LIN {X -0.027,Y -225.193,Z 1512.224,A 0.000,B 0.000,C 90.000,E1 40.334} C_DIS
LIN {X 0.094,Y -218.602,Z 1512.207,A 0.000,B 0.000,C 90.000,E1 37.237} C_DIS
LIN {X 0.128,Y -212.681,Z 1512.190,A 0.000,B 0.000,C 90.000,E1 34.119} C_DIS
LIN {X 0.027,Y -206.125,Z 1512.168,A 0.000,B 0.000,C 90.000,E1 30.207} C_DIS
LIN {X -0.041,Y -200.324,Z 1512.146,A 0.000,B 0.000,C 90.000,E1 26.232} C_DIS
LIN {X 0.082,Y -195.443,Z 1512.123,A 0.000,B 0.000,C 90.000,E1 22.153} C_DIS
LIN {X -0.062,Y -191.314,Z 1512.100,A 0.000,B 0.000,C 90.000,E1 18.109} C_DIS
LIN {X 0.065,Y -187.294,Z 1512.073,A 0.000,B 0.000,C 90.000,E1 13.119} C_DIS
LIN {X 0.047,Y -183.991,Z 1512.041,A 0.000,B 0.000,C 90.000,E1 7.296} C_DIS
LIN {X 0.026,Y -182.029,Z 1511.993,A 0.000,B 0.000,C 90.000,E1 358.682} C_DIS
LIN {X -0.047,Y -182.890,Z 1511.951,A 0.000,B 0.000,C 90.000,E1 351.141} C_DIS
LIN {X -0.073,Y -185.382,Z 1511.918,A 0.000,B 0.000,C 90.000,E1 345.283} C_DIS
LIN {X 0.069,Y -188.835,Z 1511.890,A 0.000,B 0.000,C 90.000,E1 340.242} C_DIS
LIN {X 0.097,Y -192.632,Z 1511.867,A 0.000,B 0.000,C 90.000,E1 336.102} C_DIS
LIN {X 0.032,Y -197.354,Z 1511.845,A 0.000,B 0.000,C 90.000,E1 332.025} C_DIS
LIN {X -0.004,Y -201.753,Z 1511.827,A 0.000,B 0.000,C 90.000,E1 328.791} C_DIS
LIN {X -0.067,Y -206.915,Z 1511.809,A 0.000,B 0.000,C 90.000,E1 325.595} C_DIS
LIN {X 0.012,Y -212.787,Z 1511.791,A 0.000,B 0.000,C 90.000,E1 322.396} C_DIS
LIN {X 0.031,Y -219.487,Z 1511.774,A 0.000,B 0.000,C 90.000,E1 319.256} C_DIS
LIN {X -0.081,Y -228.037,Z 1511.754,A 0.000,B 0.000,C 90.000,E1 315.810} C_DIS
LIN {X -0.043,Y -236.681,Z 1511.738,A 0.000,B 0.000,C 90.000,E1 312.771} C_DIS
LIN {X -0.083,Y -246.539,Z 1511.721,A 0.000,B 0.000,C 90.000,E1 309.806} C_DIS
LIN {X -0.058,Y -253.422,Z 1511.711,A 0.000,B 0.000,C 90.000,E1 307.971} C_DIS
LIN {X -0.074,Y -261.276,Z 1511.701,A 0.000,B 0.000,C 90.000,E1 306.171} C_DIS
LIN {X -0.032,Y -268.244,Z 1511.693,A 0.000,B 0.000,C 90.000,E1 304.739} C_DIS
LIN {X 0.169,Y -275.984,Z 1511.685,A 0.000,B 0.000,C 90.000,E1 303.293} C_DIS
LIN {X 0.012,Y -288.868,Z 1511.674,A 0.000,B 0.000,C 90.000,E1 301.258} C_DIS
LIN {X -0.059,Y -303.145,Z 1511.662,A 0.000,B 0.000,C 90.000,E1 299.255} C_DIS
LIN {X 0.162,Y -318.859,Z 1511.652,A 0.000,B 0.000,C 90.000,E1 297.257} C_DIS
LIN {X 0.039,Y -342.911,Z 1511.637,A 0.000,B 0.000,C 90.000,E1 294.591} C_DIS
LIN {X 0.109,Y -358.996,Z 1511.627,A 0.000,B 0.000,C 90.000,E1 292.898} C_DIS
LIN {X 0.010,Y -372.297,Z 1511.620,A 0.000,B 0.000,C 90.000,E1 291.535} C_DIS
LIN {X 0.017,Y -382.747,Z 1511.614,A 0.000,B 0.000,C 90.000,E1 290.429} C_DIS
LIN {X -0.118,Y -392.921,Z 1511.607,A 0.000,B 0.000,C 90.000,E1 289.322} C_DIS
LIN {X -0.060,Y -402.520,Z 1511.601,A 0.000,B 0.000,C 90.000,E1 288.181} C_DIS
LIN {X 0.022,Y -409.127,Z 1511.596,A 0.000,B 0.000,C 90.000,E1 287.330} C_DIS
LIN {X 0.049,Y -415.053,Z 1511.592,A 0.000,B 0.000,C 90.000,E1 286.496} C_DIS
LIN {X 0.127,Y -420.270,Z 1511.587,A 0.000,B 0.000,C 90.000,E1 285.662} C_DIS
LIN {X 0.000,Y -423.330,Z 1511.584,A 0.000,B 0.000,C 90.000,E1 285.134} C_DIS
LIN {X 0.162,Y -427.242,Z 1511.580,A 0.000,B 0.000,C 90.000,E1 284.300} C_DIS
LIN {X -0.166,Y -430.462,Z 1511.575,A 0.000,B 0.000,C 90.000,E1 283.536} C_DIS
LIN {X -0.227,Y -432.118,Z 1511.572,A 0.000,B 0.000,C 90.000,E1 283.008} C_DIS
LIN {X 0.234,Y -433.418,Z 1511.569,A 0.000,B 0.000,C 90.000,E1 282.411} C_DIS
LIN {X 0.098,Y -434.287,Z 1511.566,A 0.000,B 0.000,C 90.000,E1 281.895} C_DIS
LIN {X 0.060,Y -434.706,Z 1511.563,A 0.000,B 0.000,C 90.000,E1 281.366} C_DIS
LIN {X 0.027,Y -434.628,Z 1511.560,A 0.000,B 0.000,C 90.000,E1 280.838} C_DIS
LIN {X -0.006,Y -433.917,Z 1511.557,A 0.000,B 0.000,C 90.000,E1 280.310} C_DIS
LIN {X -0.116,Y -432.707,Z 1511.554,A 0.000,B 0.000,C 90.000,E1 279.792} C_DIS
LIN {X -0.155,Y -430.824,Z 1511.551,A 0.000,B 0.000,C 90.000,E1 279.265} C_DIS
LIN {X 0.154,Y -428.183,Z 1511.548,A 0.000,B 0.000,C 90.000,E1 278.690} C_DIS
LIN {X 0.083,Y -424.707,Z 1511.545,A 0.000,B 0.000,C 90.000,E1 278.163} C_DIS
LIN {X -0.065,Y -420.373,Z 1511.542,A 0.000,B 0.000,C 90.000,E1 277.644} C_DIS
LIN {X 0.182,Y -414.947,Z 1511.539,A 0.000,B 0.000,C 90.000,E1 277.068} C_DIS
LIN {X -0.099,Y -408.967,Z 1511.537,A 0.000,B 0.000,C 90.000,E1 276.606} C_DIS
LIN {X -0.009,Y -402.725,Z 1511.534,A 0.000,B 0.000,C 90.000,E1 276.144} C_DIS
LIN {X 0.054,Y -396.391,Z 1511.532,A 0.000,B 0.000,C 90.000,E1 275.739} C_DIS
LIN {X -0.021,Y -389.878,Z 1511.530,A 0.000,B 0.000,C 90.000,E1 275.391} C_DIS
LIN {X 0.072,Y -383.135,Z 1511.528,A 0.000,B 0.000,C 90.000,E1 275.049} C_DIS
LIN {X -0.084,Y -373.272,Z 1511.526,A 0.000,B 0.000,C 90.000,E1 274.645} C_DIS
LIN {X -0.080,Y -357.522,Z 1511.522,A 0.000,B 0.000,C 90.000,E1 274.012} C_DIS
LIN {X 0.125,Y -344.511,Z 1511.520,A 0.000,B 0.000,C 90.000,E1 273.498} C_DIS
LIN {X -0.002,Y -331.363,Z 1511.517,A 0.000,B 0.000,C 90.000,E1 273.094} C_DIS
LIN {X 0.011,Y -321.220,Z 1511.516,A 0.000,B 0.000,C 90.000,E1 272.808} C_DIS
LIN {X 0.022,Y -314.381,Z 1511.515,A 0.000,B 0.000,C 90.000,E1 272.636} C_DIS
LIN {X 0.092,Y -302.749,Z 1511.513,A 0.000,B 0.000,C 90.000,E1 272.407} C_DIS
LIN {X 0.053,Y -294.444,Z 1511.513,A 0.000,B 0.000,C 90.000,E1 272.293} C_DIS
LIN {X -0.020,Y -280.477,Z 1511.512,A 0.000,B 0.000,C 90.000,E1 272.178} C_DIS
LIN {X -0.124,Y -275.438,Z 1511.512,A 0.000,B 0.000,C 90.000,E1 272.178} C_DIS
LIN {X 0.066,Y -181.239,Z 1511.512,A 0.000,B 0.000,C 90.000,E1 272.121} C_DIS
LIN {X 0.075,Y -181.574,Z 1511.502,A 0.000,B 0.000,C 90.000,E1 270.401} C_DIS
LIN {X 0.051,Y -180.906,Z 1511.474,A 0.000,B 0.000,C 90.000,E1 265.355} C_DIS
LIN {X -0.055,Y -180.690,Z 1511.470,A 0.000,B 0.000,C 90.000,E1 264.546} C_DIS
LIN {X 0.024,Y -178.774,Z 1511.441,A 0.000,B 0.000,C 90.000,E1 259.454} C_DIS
LIN {X -0.074,Y -175.820,Z 1511.413,A 0.000,B 0.000,C 90.000,E1 254.393} C_DIS
LIN {X -0.073,Y -172.007,Z 1511.385,A 0.000,B 0.000,C 90.000,E1 249.263} C_DIS
LIN {X -0.096,Y -171.426,Z 1511.380,A 0.000,B 0.000,C 90.000,E1 248.411} C_DIS
LIN {X -0.041,Y -167.663,Z 1511.356,A 0.000,B 0.000,C 90.000,E1 244.076} C_DIS
LIN {X -0.100,Y -166.333,Z 1511.346,A 0.000,B 0.000,C 90.000,E1 242.359} C_DIS
LIN {X 0.032,Y -163.072,Z 1511.327,A 0.000,B 0.000,C 90.000,E1 238.820} C_DIS
LIN {X -0.056,Y -161.011,Z 1511.312,A 0.000,B 0.000,C 90.000,E1 236.215} C_DIS
LIN {X 0.054,Y -157.754,Z 1511.292,A 0.000,B 0.000,C 90.000,E1 232.637} C_DIS
LIN {X -0.007,Y -155.792,Z 1511.278,A 0.000,B 0.000,C 90.000,E1 229.989} C_DIS
LIN {X 0.047,Y -152.046,Z 1511.253,A 0.000,B 0.000,C 90.000,E1 225.486} C_DIS
LIN {X 0.064,Y -150.295,Z 1511.238,A 0.000,B 0.000,C 90.000,E1 222.771} C_DIS
LIN {X -0.010,Y -147.041,Z 1511.213,A 0.000,B 0.000,C 90.000,E1 218.257} C_DIS
LIN {X -0.018,Y -145.622,Z 1511.197,A 0.000,B 0.000,C 90.000,E1 215.518} C_DIS
LIN {X -0.018,Y -143.006,Z 1511.172,A 0.000,B 0.000,C 90.000,E1 210.924} C_DIS
LIN {X 0.039,Y -141.632,Z 1511.151,A 0.000,B 0.000,C 90.000,E1 207.206} C_DIS
LIN {X -0.036,Y -139.436,Z 1511.115,A 0.000,B 0.000,C 90.000,E1 200.737} C_DIS
LIN {X 0.018,Y -139.167,Z 1511.105,A 0.000,B 0.000,C 90.000,E1 198.852} C_DIS
LIN {X 0.051,Y -138.316,Z 1511.053,A 0.000,B 0.000,C 90.000,E1 189.500} C_DIS
LIN {X 0.063,Y -139.475,Z 1511.006,A 0.000,B 0.000,C 90.000,E1 181.088} C_DIS
LIN {X 0.004,Y -141.054,Z 1510.975,A 0.000,B 0.000,C 90.000,E1 175.527} C_DIS
LIN {X -0.042,Y -142.426,Z 1510.960,A 0.000,B 0.000,C 90.000,E1 172.761} C_DIS
LIN {X 0.019,Y -144.663,Z 1510.934,A 0.000,B 0.000,C 90.000,E1 168.117} C_DIS
LIN {X 0.002,Y -147.246,Z 1510.914,A 0.000,B 0.000,C 90.000,E1 164.448} C_DIS
LIN {X 0.021,Y -150.563,Z 1510.888,A 0.000,B 0.000,C 90.000,E1 159.880} C_DIS
LIN {X -0.041,Y -154.032,Z 1510.868,A 0.000,B 0.000,C 90.000,E1 156.282} C_DIS
LIN {X 0.028,Y -157.448,Z 1510.848,A 0.000,B 0.000,C 90.000,E1 152.666} C_DIS
LIN {X -0.023,Y -161.665,Z 1510.828,A 0.000,B 0.000,C 90.000,E1 149.125} C_DIS
LIN {X -0.006,Y -165.861,Z 1510.809,A 0.000,B 0.000,C 90.000,E1 145.595} C_DIS
LIN {X -0.015,Y -170.837,Z 1510.789,A 0.000,B 0.000,C 90.000,E1 142.110} C_DIS
LIN {X 0.032,Y -175.706,Z 1510.770,A 0.000,B 0.000,C 90.000,E1 138.647} C_DIS
LIN {X 0.023,Y -181.319,Z 1510.751,A 0.000,B 0.000,C 90.000,E1 135.243} C_DIS
LIN {X -0.105,Y -186.803,Z 1510.733,A 0.000,B 0.000,C 90.000,E1 131.919} C_DIS
LIN {X -0.035,Y -191.393,Z 1510.719,A 0.000,B 0.000,C 90.000,E1 129.402} C_DIS
LIN {X 0.048,Y -197.238,Z 1510.701,A 0.000,B 0.000,C 90.000,E1 126.091} C_DIS
LIN {X -0.029,Y -200.515,Z 1510.692,A 0.000,B 0.000,C 90.000,E1 124.485} C_DIS
LIN {X -0.003,Y -202.086,Z 1510.687,A 0.000,B 0.000,C 90.000,E1 123.579} C_DIS
LIN {X -0.056,Y -315.409,Z 1510.687,A 0.000,B 0.000,C 90.000,E1 123.579} C_DIS
LIN {X -0.208,Y -317.705,Z 1510.686,A 0.000,B 0.000,C 90.000,E1 123.579} C_DIS
LIN {X -0.007,Y -321.821,Z 1510.685,A 0.000,B 0.000,C 90.000,E1 123.372} C_DIS
LIN {X -0.072,Y -324.135,Z 1510.684,A 0.000,B 0.000,C 90.000,E1 123.214} C_DIS
LIN {X -0.110,Y -327.305,Z 1510.683,A 0.000,B 0.000,C 90.000,E1 122.880} C_DIS
LIN {X 0.123,Y -329.269,Z 1510.681,A 0.000,B 0.000,C 90.000,E1 122.546} C_DIS
LIN {X 0.079,Y -330.805,Z 1510.679,A 0.000,B 0.000,C 90.000,E1 122.260} C_DIS
LIN {X -0.056,Y -336.858,Z 1510.671,A 0.000,B 0.000,C 90.000,E1 120.718} C_DIS
LIN {X 0.206,Y -348.526,Z 1510.655,A 0.000,B 0.000,C 90.000,E1 117.897} C_DIS
LIN {X 0.014,Y -361.623,Z 1510.640,A 0.000,B 0.000,C 90.000,E1 115.207} C_DIS
LIN {X 0.213,Y -376.269,Z 1510.625,A 0.000,B 0.000,C 90.000,E1 112.514} C_DIS
LIN {X -0.101,Y -390.685,Z 1510.612,A 0.000,B 0.000,C 90.000,E1 110.248} C_DIS
LIN {X -0.201,Y -406.522,Z 1510.600,A 0.000,B 0.000,C 90.000,E1 108.000} C_DIS
LIN {X -0.164,Y -423.889,Z 1510.588,A 0.000,B 0.000,C 90.000,E1 105.788} C_DIS
LIN {X 0.203,Y -442.903,Z 1510.576,A 0.000,B 0.000,C 90.000,E1 103.592} C_DIS
LIN {X 0.100,Y -462.926,Z 1510.564,A 0.000,B 0.000,C 90.000,E1 101.591} C_DIS
LIN {X -0.208,Y -486.084,Z 1510.553,A 0.000,B 0.000,C 90.000,E1 99.557} C_DIS
LIN {X 0.021,Y -491.185,Z 1510.551,A 0.000,B 0.000,C 90.000,E1 99.095} C_DIS
LIN {X 0.195,Y -493.088,Z 1510.549,A 0.000,B 0.000,C 90.000,E1 98.859} C_DIS
LIN {X 0.103,Y -494.734,Z 1510.548,A 0.000,B 0.000,C 90.000,E1 98.624} C_DIS
LIN {X -0.064,Y -495.964,Z 1510.547,A 0.000,B 0.000,C 90.000,E1 98.398} C_DIS
LIN {X 0.257,Y -497.454,Z 1510.544,A 0.000,B 0.000,C 90.000,E1 97.871} C_DIS
LIN {X 0.023,Y -497.876,Z 1510.541,A 0.000,B 0.000,C 90.000,E1 97.409} C_DIS
LIN {X -0.204,Y -497.304,Z 1510.538,A 0.000,B 0.000,C 90.000,E1 96.947} C_DIS
LIN {X 0.066,Y -495.646,Z 1510.536,A 0.000,B 0.000,C 90.000,E1 96.429} C_DIS
LIN {X -0.075,Y -494.316,Z 1510.534,A 0.000,B 0.000,C 90.000,E1 96.201} C_DIS
LIN {X 0.147,Y -484.472,Z 1510.526,A 0.000,B 0.000,C 90.000,E1 94.702} C_DIS
LIN {X 0.127,Y -475.397,Z 1510.518,A 0.000,B 0.000,C 90.000,E1 93.212} C_DIS
LIN {X 0.164,Y -467.375,Z 1510.511,A 0.000,B 0.000,C 90.000,E1 91.949} C_DIS
LIN {X 0.075,Y -458.921,Z 1510.504,A 0.000,B 0.000,C 90.000,E1 90.688} C_DIS
LIN {X 0.077,Y -448.386,Z 1510.495,A 0.000,B 0.000,C 90.000,E1 89.141} C_DIS
LIN {X 0.174,Y -439.501,Z 1510.488,A 0.000,B 0.000,C 90.000,E1 87.822} C_DIS
LIN {X -0.011,Y -426.646,Z 1510.478,A 0.000,B 0.000,C 90.000,E1 85.988} C_DIS
LIN {X 0.029,Y -413.901,Z 1510.467,A 0.000,B 0.000,C 90.000,E1 84.090} C_DIS
LIN {X -0.149,Y -401.127,Z 1510.456,A 0.000,B 0.000,C 90.000,E1 82.186} C_DIS
LIN {X 0.010,Y -383.248,Z 1510.441,A 0.000,B 0.000,C 90.000,E1 79.342} C_DIS
LIN {X -0.122,Y -368.118,Z 1510.426,A 0.000,B 0.000,C 90.000,E1 76.756} C_DIS
LIN {X -0.157,Y -355.156,Z 1510.413,A 0.000,B 0.000,C 90.000,E1 74.393} C_DIS
LIN {X 0.101,Y -343.908,Z 1510.401,A 0.000,B 0.000,C 90.000,E1 72.236} C_DIS
LIN {X 0.199,Y -331.258,Z 1510.388,A 0.000,B 0.000,C 90.000,E1 69.752} C_DIS
LIN {X 0.092,Y -316.207,Z 1510.370,A 0.000,B 0.000,C 90.000,E1 66.613} C_DIS
LIN {X 0.011,Y -303.308,Z 1510.354,A 0.000,B 0.000,C 90.000,E1 63.717} C_DIS
LIN {X 0.118,Y -292.356,Z 1510.339,A 0.000,B 0.000,C 90.000,E1 61.051} C_DIS
LIN {X -0.036,Y -280.499,Z 1510.322,A 0.000,B 0.000,C 90.000,E1 58.043} C_DIS
LIN {X 0.083,Y -270.320,Z 1510.307,A 0.000,B 0.000,C 90.000,E1 55.261} C_DIS
LIN {X -0.091,Y -261.656,Z 1510.293,A 0.000,B 0.000,C 90.000,E1 52.844} C_DIS
LIN {X -0.077,Y -250.902,Z 1510.276,A 0.000,B 0.000,C 90.000,E1 49.622} C_DIS
LIN {X 0.098,Y -240.948,Z 1510.257,A 0.000,B 0.000,C 90.000,E1 46.296} C_DIS
LIN {X 0.053,Y -232.820,Z 1510.241,A 0.000,B 0.000,C 90.000,E1 43.338} C_DIS
LIN {X -0.004,Y -225.479,Z 1510.224,A 0.000,B 0.000,C 90.000,E1 40.334} C_DIS
LIN {X -0.050,Y -218.895,Z 1510.207,A 0.000,B 0.000,C 90.000,E1 37.282} C_DIS
LIN {X -0.133,Y -212.982,Z 1510.190,A 0.000,B 0.000,C 90.000,E1 34.199} C_DIS
LIN {X 0.070,Y -206.391,Z 1510.168,A 0.000,B 0.000,C 90.000,E1 30.207} C_DIS
LIN {X 0.009,Y -200.601,Z 1510.146,A 0.000,B 0.000,C 90.000,E1 26.232} C_DIS
LIN {X -0.042,Y -195.697,Z 1510.123,A 0.000,B 0.000,C 90.000,E1 22.206} C_DIS
LIN {X -0.058,Y -191.585,Z 1510.101,A 0.000,B 0.000,C 90.000,E1 18.127} C_DIS
LIN {X -0.044,Y -187.555,Z 1510.073,A 0.000,B 0.000,C 90.000,E1 13.175} C_DIS
LIN {X -0.054,Y -184.269,Z 1510.041,A 0.000,B 0.000,C 90.000,E1 7.352} C_DIS
LIN {X 0.027,Y -182.284,Z 1509.993,A 0.000,B 0.000,C 90.000,E1 358.682} C_DIS
LIN {X -0.032,Y -183.151,Z 1509.951,A 0.000,B 0.000,C 90.000,E1 351.141} C_DIS
LIN {X -0.046,Y -185.605,Z 1509.918,A 0.000,B 0.000,C 90.000,E1 345.283} C_DIS
LIN {X 0.104,Y -189.040,Z 1509.890,A 0.000,B 0.000,C 90.000,E1 340.242} C_DIS
LIN {X -0.115,Y -192.834,Z 1509.867,A 0.000,B 0.000,C 90.000,E1 336.177} C_DIS
LIN {X 0.081,Y -197.507,Z 1509.845,A 0.000,B 0.000,C 90.000,E1 332.025} C_DIS
LIN {X 0.014,Y -203.113,Z 1509.822,A 0.000,B 0.000,C 90.000,E1 327.995} C_DIS
LIN {X -0.073,Y -208.455,Z 1509.804,A 0.000,B 0.000,C 90.000,E1 324.815} C_DIS
LIN {X 0.044,Y -214.529,Z 1509.787,A 0.000,B 0.000,C 90.000,E1 321.618} C_DIS
LIN {X 0.077,Y -221.411,Z 1509.770,A 0.000,B 0.000,C 90.000,E1 318.485} C_DIS
LIN {X 0.086,Y -229.191,Z 1509.752,A 0.000,B 0.000,C 90.000,E1 315.405} C_DIS
LIN {X 0.001,Y -237.989,Z 1509.736,A 0.000,B 0.000,C 90.000,E1 312.405} C_DIS
LIN {X 0.003,Y -247.980,Z 1509.719,A 0.000,B 0.000,C 90.000,E1 309.439} C_DIS
LIN {X 0.058,Y -255.024,Z 1509.709,A 0.000,B 0.000,C 90.000,E1 307.604} C_DIS
LIN {X 0.065,Y -263.042,Z 1509.699,A 0.000,B 0.000,C 90.000,E1 305.804} C_DIS
LIN {X -0.024,Y -270.146,Z 1509.691,A 0.000,B 0.000,C 90.000,E1 304.405} C_DIS
LIN {X -0.087,Y -280.099,Z 1509.681,A 0.000,B 0.000,C 90.000,E1 302.673} C_DIS
LIN {X 0.073,Y -293.344,Z 1509.670,A 0.000,B 0.000,C 90.000,E1 300.590} C_DIS
LIN {X -0.058,Y -308.047,Z 1509.659,A 0.000,B 0.000,C 90.000,E1 298.615} C_DIS
LIN {X -0.093,Y -332.075,Z 1509.643,A 0.000,B 0.000,C 90.000,E1 295.796} C_DIS
LIN {X -0.061,Y -350.991,Z 1509.632,A 0.000,B 0.000,C 90.000,E1 293.770} C_DIS
LIN {X 0.180,Y -364.572,Z 1509.624,A 0.000,B 0.000,C 90.000,E1 292.333} C_DIS
LIN {X -0.110,Y -375.152,Z 1509.618,A 0.000,B 0.000,C 90.000,E1 291.280} C_DIS
LIN {X -0.135,Y -385.509,Z 1509.612,A 0.000,B 0.000,C 90.000,E1 290.174} C_DIS
LIN {X -0.001,Y -395.496,Z 1509.606,A 0.000,B 0.000,C 90.000,E1 289.033} C_DIS
LIN {X 0.217,Y -404.974,Z 1509.599,A 0.000,B 0.000,C 90.000,E1 287.873} C_DIS
LIN {X -0.184,Y -411.370,Z 1509.595,A 0.000,B 0.000,C 90.000,E1 287.094} C_DIS
LIN {X -0.144,Y -417.125,Z 1509.590,A 0.000,B 0.000,C 90.000,E1 286.260} C_DIS
LIN {X -0.042,Y -422.082,Z 1509.586,A 0.000,B 0.000,C 90.000,E1 285.426} C_DIS
LIN {X -0.159,Y -424.990,Z 1509.583,A 0.000,B 0.000,C 90.000,E1 284.898} C_DIS
LIN {X 0.012,Y -428.722,Z 1509.578,A 0.000,B 0.000,C 90.000,E1 284.064} C_DIS
LIN {X -0.061,Y -430.824,Z 1509.575,A 0.000,B 0.000,C 90.000,E1 283.536} C_DIS
LIN {X -0.120,Y -432.509,Z 1509.572,A 0.000,B 0.000,C 90.000,E1 283.008} C_DIS
LIN {X -0.172,Y -433.869,Z 1509.569,A 0.000,B 0.000,C 90.000,E1 282.479} C_DIS
LIN {X -0.214,Y -434.795,Z 1509.566,A 0.000,B 0.000,C 90.000,E1 281.951} C_DIS
LIN {X 0.176,Y -435.234,Z 1509.563,A 0.000,B 0.000,C 90.000,E1 281.366} C_DIS
LIN {X 0.147,Y -435.188,Z 1509.560,A 0.000,B 0.000,C 90.000,E1 280.838} C_DIS
LIN {X 0.117,Y -434.530,Z 1509.557,A 0.000,B 0.000,C 90.000,E1 280.310} C_DIS
LIN {X 0.009,Y -433.338,Z 1509.554,A 0.000,B 0.000,C 90.000,E1 279.792} C_DIS
LIN {X -0.027,Y -431.499,Z 1509.551,A 0.000,B 0.000,C 90.000,E1 279.265} C_DIS
LIN {X 0.162,Y -430.313,Z 1509.550,A 0.000,B 0.000,C 90.000,E1 278.973} C_DIS
LIN {X 0.041,Y -427.294,Z 1509.547,A 0.000,B 0.000,C 90.000,E1 278.454} C_DIS
LIN {X -0.094,Y -423.434,Z 1509.544,A 0.000,B 0.000,C 90.000,E1 277.936} C_DIS
LIN {X -0.190,Y -418.628,Z 1509.541,A 0.000,B 0.000,C 90.000,E1 277.409} C_DIS
LIN {X 0.196,Y -412.957,Z 1509.538,A 0.000,B 0.000,C 90.000,E1 276.834} C_DIS
LIN {X 0.072,Y -406.867,Z 1509.535,A 0.000,B 0.000,C 90.000,E1 276.372} C_DIS
LIN {X -0.085,Y -400.503,Z 1509.533,A 0.000,B 0.000,C 90.000,E1 275.967} C_DIS
LIN {X 0.065,Y -394.051,Z 1509.531,A 0.000,B 0.000,C 90.000,E1 275.568} C_DIS
LIN {X -0.185,Y -384.215,Z 1509.528,A 0.000,B 0.000,C 90.000,E1 275.106} C_DIS
LIN {X 0.016,Y -374.314,Z 1509.526,A 0.000,B 0.000,C 90.000,E1 274.645} C_DIS
LIN {X 0.004,Y -358.544,Z 1509.522,A 0.000,B 0.000,C 90.000,E1 274.012} C_DIS
LIN {X -0.134,Y -345.601,Z 1509.520,A 0.000,B 0.000,C 90.000,E1 273.555} C_DIS
LIN {X 0.057,Y -332.304,Z 1509.517,A 0.000,B 0.000,C 90.000,E1 273.094} C_DIS
LIN {X -0.129,Y -318.650,Z 1509.515,A 0.000,B 0.000,C 90.000,E1 272.751} C_DIS
LIN {X -0.141,Y -307.348,Z 1509.514,A 0.000,B 0.000,C 90.000,E1 272.522} C_DIS
LIN {X 0.071,Y -295.137,Z 1509.513,A 0.000,B 0.000,C 90.000,E1 272.293} C_DIS
LIN {X 0.004,Y -280.690,Z 1509.512,A 0.000,B 0.000,C 90.000,E1 272.178} C_DIS
LIN {X -0.098,Y -276.198,Z 1509.512,A 0.000,B 0.000,C 90.000,E1 272.178} C_DIS
LIN {X 0.084,Y -181.238,Z 1509.512,A 0.000,B 0.000,C 90.000,E1 272.121} C_DIS
LIN {X -0.086,Y -181.573,Z 1509.502,A 0.000,B 0.000,C 90.000,E1 270.458} C_DIS
LIN {X 0.072,Y -180.906,Z 1509.474,A 0.000,B 0.000,C 90.000,E1 265.355} C_DIS
LIN {X -0.034,Y -180.693,Z 1509.470,A 0.000,B 0.000,C 90.000,E1 264.546} C_DIS
LIN {X 0.044,Y -178.778,Z 1509.442,A 0.000,B 0.000,C 90.000,E1 259.454} C_DIS
LIN {X -0.054,Y -175.824,Z 1509.413,A 0.000,B 0.000,C 90.000,E1 254.393} C_DIS
LIN {X -0.053,Y -172.012,Z 1509.385,A 0.000,B 0.000,C 90.000,E1 249.263} C_DIS
LIN {X -0.077,Y -171.432,Z 1509.380,A 0.000,B 0.000,C 90.000,E1 248.411} C_DIS
LIN {X -0.022,Y -167.668,Z 1509.356,A 0.000,B 0.000,C 90.000,E1 244.076} C_DIS
LIN {X -0.080,Y -166.341,Z 1509.346,A 0.000,B 0.000,C 90.000,E1 242.359} C_DIS
LIN {X -0.088,Y -163.077,Z 1509.327,A 0.000,B 0.000,C 90.000,E1 238.869} C_DIS
LIN {X -0.037,Y -161.017,Z 1509.312,A 0.000,B 0.000,C 90.000,E1 236.215} C_DIS
LIN {X -0.052,Y -157.760,Z 1509.293,A 0.000,B 0.000,C 90.000,E1 232.683} C_DIS
LIN {X 0.011,Y -155.798,Z 1509.278,A 0.000,B 0.000,C 90.000,E1 229.989} C_DIS
LIN {X 0.065,Y -152.050,Z 1509.253,A 0.000,B 0.000,C 90.000,E1 225.486} C_DIS
LIN {X 0.083,Y -150.300,Z 1509.238,A 0.000,B 0.000,C 90.000,E1 222.771} C_DIS
LIN {X 0.009,Y -147.046,Z 1509.213,A 0.000,B 0.000,C 90.000,E1 218.257} C_DIS
LIN {X 0.001,Y -145.625,Z 1509.197,A 0.000,B 0.000,C 90.000,E1 215.518} C_DIS
LIN {X -0.001,Y -143.009,Z 1509.172,A 0.000,B 0.000,C 90.000,E1 210.924} C_DIS
LIN {X -0.070,Y -141.635,Z 1509.151,A 0.000,B 0.000,C 90.000,E1 207.257} C_DIS
LIN {X -0.018,Y -139.437,Z 1509.115,A 0.000,B 0.000,C 90.000,E1 200.737} C_DIS
LIN {X 0.035,Y -139.169,Z 1509.105,A 0.000,B 0.000,C 90.000,E1 198.852} C_DIS
LIN {X -0.067,Y -138.317,Z 1509.053,A 0.000,B 0.000,C 90.000,E1 189.557} C_DIS
LIN {X -0.059,Y -139.474,Z 1509.006,A 0.000,B 0.000,C 90.000,E1 181.146} C_DIS
LIN {X 0.022,Y -141.051,Z 1508.975,A 0.000,B 0.000,C 90.000,E1 175.527} C_DIS
LIN {X -0.024,Y -142.422,Z 1508.960,A 0.000,B 0.000,C 90.000,E1 172.761} C_DIS
LIN {X 0.037,Y -144.658,Z 1508.934,A 0.000,B 0.000,C 90.000,E1 168.117} C_DIS
LIN {X 0.020,Y -147.241,Z 1508.914,A 0.000,B 0.000,C 90.000,E1 164.448} C_DIS
LIN {X 0.039,Y -150.558,Z 1508.888,A 0.000,B 0.000,C 90.000,E1 159.880} C_DIS
LIN {X -0.022,Y -154.026,Z 1508.868,A 0.000,B 0.000,C 90.000,E1 156.282} C_DIS
LIN {X 0.047,Y -157.441,Z 1508.848,A 0.000,B 0.000,C 90.000,E1 152.666} C_DIS
LIN {X -0.004,Y -161.656,Z 1508.828,A 0.000,B 0.000,C 90.000,E1 149.125} C_DIS
LIN {X 0.013,Y -165.851,Z 1508.809,A 0.000,B 0.000,C 90.000,E1 145.595} C_DIS
LIN {X 0.005,Y -170.827,Z 1508.790,A 0.000,B 0.000,C 90.000,E1 142.110} C_DIS
LIN {X -0.079,Y -175.696,Z 1508.770,A 0.000,B 0.000,C 90.000,E1 138.690} C_DIS
LIN {X 0.045,Y -181.309,Z 1508.751,A 0.000,B 0.000,C 90.000,E1 135.243} C_DIS
LIN {X -0.084,Y -186.792,Z 1508.733,A 0.000,B 0.000,C 90.000,E1 131.919} C_DIS
LIN {X -0.014,Y -191.383,Z 1508.719,A 0.000,B 0.000,C 90.000,E1 129.402} C_DIS
LIN {X 0.069,Y -197.226,Z 1508.701,A 0.000,B 0.000,C 90.000,E1 126.091} C_DIS
LIN {X -0.007,Y -200.503,Z 1508.692,A 0.000,B 0.000,C 90.000,E1 124.485} C_DIS
LIN {X 0.087,Y -202.041,Z 1508.687,A 0.000,B 0.000,C 90.000,E1 123.579} C_DIS
LIN {X 0.101,Y -315.676,Z 1508.687,A 0.000,B 0.000,C 90.000,E1 123.579} C_DIS
LIN {X -0.174,Y -318.465,Z 1508.686,A 0.000,B 0.000,C 90.000,E1 123.579} C_DIS
LIN {X 0.028,Y -322.062,Z 1508.685,A 0.000,B 0.000,C 90.000,E1 123.372} C_DIS
LIN {X -0.037,Y -324.270,Z 1508.684,A 0.000,B 0.000,C 90.000,E1 123.214} C_DIS
LIN {X -0.075,Y -327.351,Z 1508.683,A 0.000,B 0.000,C 90.000,E1 122.880} C_DIS
LIN {X 0.124,Y -329.310,Z 1508.681,A 0.000,B 0.000,C 90.000,E1 122.546} C_DIS
LIN {X 0.045,Y -330.839,Z 1508.679,A 0.000,B 0.000,C 90.000,E1 122.260} C_DIS
LIN {X 0.002,Y -345.818,Z 1508.659,A 0.000,B 0.000,C 90.000,E1 118.537} C_DIS
LIN {X 0.046,Y -358.590,Z 1508.643,A 0.000,B 0.000,C 90.000,E1 115.796} C_DIS
LIN {X -0.026,Y -372.885,Z 1508.629,A 0.000,B 0.000,C 90.000,E1 113.131} C_DIS
LIN {X 0.066,Y -386.964,Z 1508.616,A 0.000,B 0.000,C 90.000,E1 110.791} C_DIS
LIN {X -0.123,Y -402.440,Z 1508.603,A 0.000,B 0.000,C 90.000,E1 108.544} C_DIS
LIN {X -0.066,Y -419.416,Z 1508.591,A 0.000,B 0.000,C 90.000,E1 106.315} C_DIS
LIN {X 0.180,Y -438.015,Z 1508.579,A 0.000,B 0.000,C 90.000,E1 104.120} C_DIS
LIN {X 0.181,Y -457.892,Z 1508.567,A 0.000,B 0.000,C 90.000,E1 102.063} C_DIS
LIN {X -0.019,Y -478.331,Z 1508.557,A 0.000,B 0.000,C 90.000,E1 100.197} C_DIS
LIN {X -0.020,Y -491.191,Z 1508.551,A 0.000,B 0.000,C 90.000,E1 99.095} C_DIS
LIN {X 0.154,Y -493.066,Z 1508.549,A 0.000,B 0.000,C 90.000,E1 98.859} C_DIS
LIN {X 0.062,Y -494.693,Z 1508.548,A 0.000,B 0.000,C 90.000,E1 98.624} C_DIS
LIN {X -0.106,Y -495.906,Z 1508.547,A 0.000,B 0.000,C 90.000,E1 98.398} C_DIS
LIN {X 0.215,Y -497.371,Z 1508.544,A 0.000,B 0.000,C 90.000,E1 97.871} C_DIS
LIN {X -0.020,Y -497.773,Z 1508.541,A 0.000,B 0.000,C 90.000,E1 97.409} C_DIS
LIN {X 0.247,Y -497.180,Z 1508.538,A 0.000,B 0.000,C 90.000,E1 96.891} C_DIS
LIN {X 0.023,Y -495.497,Z 1508.536,A 0.000,B 0.000,C 90.000,E1 96.429} C_DIS
LIN {X -0.118,Y -494.151,Z 1508.534,A 0.000,B 0.000,C 90.000,E1 96.201} C_DIS
LIN {X 0.222,Y -485.849,Z 1508.528,A 0.000,B 0.000,C 90.000,E1 94.935} C_DIS
LIN {X 0.080,Y -475.233,Z 1508.518,A 0.000,B 0.000,C 90.000,E1 93.212} C_DIS
LIN {X -0.163,Y -468.859,Z 1508.512,A 0.000,B 0.000,C 90.000,E1 92.236} C_DIS
LIN {X 0.025,Y -458.750,Z 1508.504,A 0.000,B 0.000,C 90.000,E1 90.688} C_DIS
LIN {X 0.026,Y -448.246,Z 1508.495,A 0.000,B 0.000,C 90.000,E1 89.141} C_DIS
LIN {X 0.121,Y -439.360,Z 1508.488,A 0.000,B 0.000,C 90.000,E1 87.822} C_DIS
LIN {X -0.064,Y -426.561,Z 1508.478,A 0.000,B 0.000,C 90.000,E1 85.988} C_DIS
LIN {X -0.024,Y -413.870,Z 1508.467,A 0.000,B 0.000,C 90.000,E1 84.090} C_DIS
LIN {X -0.107,Y -399.296,Z 1508.455,A 0.000,B 0.000,C 90.000,E1 81.894} C_DIS
LIN {X 0.029,Y -379.803,Z 1508.438,A 0.000,B 0.000,C 90.000,E1 78.757} C_DIS
LIN {X 0.162,Y -364.867,Z 1508.423,A 0.000,B 0.000,C 90.000,E1 76.117} C_DIS
LIN {X 0.082,Y -353.568,Z 1508.411,A 0.000,B 0.000,C 90.000,E1 74.047} C_DIS
LIN {X -0.031,Y -342.331,Z 1508.400,A 0.000,B 0.000,C 90.000,E1 71.945} C_DIS
LIN {X 0.156,Y -331.250,Z 1508.388,A 0.000,B 0.000,C 90.000,E1 69.752} C_DIS
LIN {X 0.050,Y -316.171,Z 1508.370,A 0.000,B 0.000,C 90.000,E1 66.613} C_DIS
LIN {X -0.029,Y -303.269,Z 1508.354,A 0.000,B 0.000,C 90.000,E1 63.717} C_DIS
LIN {X 0.075,Y -290.989,Z 1508.337,A 0.000,B 0.000,C 90.000,E1 60.717} C_DIS
LIN {X 0.127,Y -279.235,Z 1508.320,A 0.000,B 0.000,C 90.000,E1 57.661} C_DIS
LIN {X 0.132,Y -269.126,Z 1508.305,A 0.000,B 0.000,C 90.000,E1 54.895} C_DIS
LIN {X -0.069,Y -260.537,Z 1508.292,A 0.000,B 0.000,C 90.000,E1 52.477} C_DIS
LIN {X 0.081,Y -249.938,Z 1508.274,A 0.000,B 0.000,C 90.000,E1 49.218} C_DIS
LIN {X 0.048,Y -239.093,Z 1508.253,A 0.000,B 0.000,C 90.000,E1 45.567} C_DIS
LIN {X -0.042,Y -231.130,Z 1508.237,A 0.000,B 0.000,C 90.000,E1 42.609} C_DIS
LIN {X -0.092,Y -222.345,Z 1508.216,A 0.000,B 0.000,C 90.000,E1 38.830} C_DIS
LIN {X 0.000,Y -214.642,Z 1508.194,A 0.000,B 0.000,C 90.000,E1 34.945} C_DIS
LIN {X 0.070,Y -207.880,Z 1508.172,A 0.000,B 0.000,C 90.000,E1 31.003} C_DIS
LIN {X -0.030,Y -201.949,Z 1508.150,A 0.000,B 0.000,C 90.000,E1 27.052} C_DIS
LIN {X -0.040,Y -196.849,Z 1508.128,A 0.000,B 0.000,C 90.000,E1 23.025} C_DIS
LIN {X -0.067,Y -192.605,Z 1508.105,A 0.000,B 0.000,C 90.000,E1 18.960} C_DIS
LIN {X -0.018,Y -188.421,Z 1508.078,A 0.000,B 0.000,C 90.000,E1 14.008} C_DIS
LIN {X -0.025,Y -185.312,Z 1508.050,A 0.000,B 0.000,C 90.000,E1 9.029} C_DIS
LIN {X 0.015,Y -182.839,Z 1508.008,A 0.000,B 0.000,C 90.000,E1 1.489} C_DIS
LIN {X 0.080,Y -182.845,Z 1507.965,A 0.000,B 0.000,C 90.000,E1 353.628} C_DIS
LIN {X 0.036,Y -184.978,Z 1507.927,A 0.000,B 0.000,C 90.000,E1 346.937} C_DIS
LIN {X -0.002,Y -187.977,Z 1507.900,A 0.000,B 0.000,C 90.000,E1 341.945} C_DIS
LIN {X 0.031,Y -191.387,Z 1507.877,A 0.000,B 0.000,C 90.000,E1 337.794} C_DIS
LIN {X 0.014,Y -195.696,Z 1507.854,A 0.000,B 0.000,C 90.000,E1 333.691} C_DIS
LIN {X 0.044,Y -200.877,Z 1507.831,A 0.000,B 0.000,C 90.000,E1 329.616} C_DIS
LIN {X -0.044,Y -205.813,Z 1507.813,A 0.000,B 0.000,C 90.000,E1 326.421} C_DIS
LIN {X 0.053,Y -211.512,Z 1507.796,A 0.000,B 0.000,C 90.000,E1 323.210} C_DIS
LIN {X 0.038,Y -217.987,Z 1507.778,A 0.000,B 0.000,C 90.000,E1 320.070} C_DIS
LIN {X -0.101,Y -226.271,Z 1507.759,A 0.000,B 0.000,C 90.000,E1 316.620} C_DIS
LIN {X 0.005,Y -235.808,Z 1507.740,A 0.000,B 0.000,C 90.000,E1 313.176} C_DIS
LIN {X 0.107,Y -245.499,Z 1507.723,A 0.000,B 0.000,C 90.000,E1 310.172} C_DIS
LIN {X -0.063,Y -253.639,Z 1507.711,A 0.000,B 0.000,C 90.000,E1 308.016} C_DIS
LIN {X -0.080,Y -261.434,Z 1507.701,A 0.000,B 0.000,C 90.000,E1 306.217} C_DIS
LIN {X 0.087,Y -270.185,Z 1507.691,A 0.000,B 0.000,C 90.000,E1 304.405} C_DIS
LIN {X 0.029,Y -280.069,Z 1507.682,A 0.000,B 0.000,C 90.000,E1 302.673} C_DIS
LIN {X 0.044,Y -293.236,Z 1507.670,A 0.000,B 0.000,C 90.000,E1 300.620} C_DIS
LIN {X 0.040,Y -305.304,Z 1507.661,A 0.000,B 0.000,C 90.000,E1 298.949} C_DIS
LIN {X -0.125,Y -329.442,Z 1507.645,A 0.000,B 0.000,C 90.000,E1 296.104} C_DIS
LIN {X -0.086,Y -348.238,Z 1507.634,A 0.000,B 0.000,C 90.000,E1 294.079} C_DIS
LIN {X 0.005,Y -364.543,Z 1507.624,A 0.000,B 0.000,C 90.000,E1 292.386} C_DIS
LIN {X 0.110,Y -375.061,Z 1507.618,A 0.000,B 0.000,C 90.000,E1 291.280} C_DIS
LIN {X 0.159,Y -385.329,Z 1507.612,A 0.000,B 0.000,C 90.000,E1 290.174} C_DIS
LIN {X -0.144,Y -395.417,Z 1507.606,A 0.000,B 0.000,C 90.000,E1 289.087} C_DIS
LIN {X -0.059,Y -404.960,Z 1507.600,A 0.000,B 0.000,C 90.000,E1 287.946} C_DIS
LIN {X 0.054,Y -411.409,Z 1507.595,A 0.000,B 0.000,C 90.000,E1 287.094} C_DIS
LIN {X 0.098,Y -417.212,Z 1507.590,A 0.000,B 0.000,C 90.000,E1 286.260} C_DIS
LIN {X 0.203,Y -422.268,Z 1507.586,A 0.000,B 0.000,C 90.000,E1 285.426} C_DIS
LIN {X 0.089,Y -425.200,Z 1507.583,A 0.000,B 0.000,C 90.000,E1 284.898} C_DIS
LIN {X -0.152,Y -428.963,Z 1507.578,A 0.000,B 0.000,C 90.000,E1 284.120} C_DIS
LIN {X 0.194,Y -431.121,Z 1507.575,A 0.000,B 0.000,C 90.000,E1 283.536} C_DIS
LIN {X 0.139,Y -432.866,Z 1507.572,A 0.000,B 0.000,C 90.000,E1 283.008} C_DIS
LIN {X 0.088,Y -434.282,Z 1507.569,A 0.000,B 0.000,C 90.000,E1 282.479} C_DIS
LIN {X 0.048,Y -435.252,Z 1507.566,A 0.000,B 0.000,C 90.000,E1 281.951} C_DIS
LIN {X 0.015,Y -435.739,Z 1507.563,A 0.000,B 0.000,C 90.000,E1 281.422} C_DIS
LIN {X -0.013,Y -435.734,Z 1507.561,A 0.000,B 0.000,C 90.000,E1 280.894} C_DIS
LIN {X -0.041,Y -435.159,Z 1507.558,A 0.000,B 0.000,C 90.000,E1 280.366} C_DIS
LIN {X -0.145,Y -434.029,Z 1507.555,A 0.000,B 0.000,C 90.000,E1 279.849} C_DIS
LIN {X -0.177,Y -432.251,Z 1507.552,A 0.000,B 0.000,C 90.000,E1 279.321} C_DIS
LIN {X 0.014,Y -431.106,Z 1507.550,A 0.000,B 0.000,C 90.000,E1 279.029} C_DIS
LIN {X -0.103,Y -428.178,Z 1507.547,A 0.000,B 0.000,C 90.000,E1 278.511} C_DIS
LIN {X 0.188,Y -424.378,Z 1507.544,A 0.000,B 0.000,C 90.000,E1 277.936} C_DIS
LIN {X 0.094,Y -419.648,Z 1507.541,A 0.000,B 0.000,C 90.000,E1 277.409} C_DIS
LIN {X 0.036,Y -414.063,Z 1507.538,A 0.000,B 0.000,C 90.000,E1 276.891} C_DIS
LIN {X -0.103,Y -407.987,Z 1507.536,A 0.000,B 0.000,C 90.000,E1 276.429} C_DIS
LIN {X 0.140,Y -401.735,Z 1507.533,A 0.000,B 0.000,C 90.000,E1 275.967} C_DIS
LIN {X -0.131,Y -395.286,Z 1507.531,A 0.000,B 0.000,C 90.000,E1 275.625} C_DIS
LIN {X -0.075,Y -388.764,Z 1507.529,A 0.000,B 0.000,C 90.000,E1 275.277} C_DIS
LIN {X -0.045,Y -378.894,Z 1507.527,A 0.000,B 0.000,C 90.000,E1 274.821} C_DIS
LIN {X -0.122,Y -366.106,Z 1507.524,A 0.000,B 0.000,C 90.000,E1 274.302} C_DIS
LIN {X 0.051,Y -353.351,Z 1507.521,A 0.000,B 0.000,C 90.000,E1 273.784} C_DIS
LIN {X 0.093,Y -344.053,Z 1507.519,A 0.000,B 0.000,C 90.000,E1 273.440} C_DIS
LIN {X 0.013,Y -330.681,Z 1507.517,A 0.000,B 0.000,C 90.000,E1 273.037} C_DIS
LIN {X 0.060,Y -320.518,Z 1507.515,A 0.000,B 0.000,C 90.000,E1 272.751} C_DIS
LIN {X 0.018,Y -309.548,Z 1507.514,A 0.000,B 0.000,C 90.000,E1 272.522} C_DIS
LIN {X -0.077,Y -297.785,Z 1507.513,A 0.000,B 0.000,C 90.000,E1 272.350} C_DIS
LIN {X -0.060,Y -286.837,Z 1507.512,A 0.000,B 0.000,C 90.000,E1 272.236} C_DIS
LIN {X -0.091,Y -275.116,Z 1507.512,A 0.000,B 0.000,C 90.000,E1 272.178} C_DIS
LIN {X 0.087,Y -181.238,Z 1507.512,A 0.000,B 0.000,C 90.000,E1 272.121} C_DIS
LIN {X 0.009,Y -181.574,Z 1507.501,A 0.000,B 0.000,C 90.000,E1 270.115} C_DIS
LIN {X -0.002,Y -180.875,Z 1507.473,A 0.000,B 0.000,C 90.000,E1 265.065} C_DIS
LIN {X 0.054,Y -178.993,Z 1507.444,A 0.000,B 0.000,C 90.000,E1 259.982} C_DIS
LIN {X 0.065,Y -177.981,Z 1507.435,A 0.000,B 0.000,C 90.000,E1 258.285} C_DIS
LIN {X 0.036,Y -175.625,Z 1507.411,A 0.000,B 0.000,C 90.000,E1 254.047} C_DIS
LIN {X 0.095,Y -172.346,Z 1507.388,A 0.000,B 0.000,C 90.000,E1 249.752} C_DIS
LIN {X 0.047,Y -171.124,Z 1507.378,A 0.000,B 0.000,C 90.000,E1 248.050} C_DIS
LIN {X -0.066,Y -167.434,Z 1507.354,A 0.000,B 0.000,C 90.000,E1 243.768} C_DIS
LIN {X 0.016,Y -166.830,Z 1507.349,A 0.000,B 0.000,C 90.000,E1 242.871} C_DIS
LIN {X -0.067,Y -162.812,Z 1507.325,A 0.000,B 0.000,C 90.000,E1 238.535} C_DIS
LIN {X -0.003,Y -161.498,Z 1507.315,A 0.000,B 0.000,C 90.000,E1 236.755} C_DIS
LIN {X -0.049,Y -157.495,Z 1507.291,A 0.000,B 0.000,C 90.000,E1 232.351} C_DIS
LIN {X -0.015,Y -155.515,Z 1507.276,A 0.000,B 0.000,C 90.000,E1 229.666} C_DIS
LIN {X 0.034,Y -151.815,Z 1507.251,A 0.000,B 0.000,C 90.000,E1 225.162} C_DIS
LIN {X 0.047,Y -150.028,Z 1507.236,A 0.000,B 0.000,C 90.000,E1 222.447} C_DIS
LIN {X -0.038,Y -146.848,Z 1507.211,A 0.000,B 0.000,C 90.000,E1 217.935} C_DIS
LIN {X -0.020,Y -145.431,Z 1507.195,A 0.000,B 0.000,C 90.000,E1 215.185} C_DIS
LIN {X -0.024,Y -142.854,Z 1507.170,A 0.000,B 0.000,C 90.000,E1 210.590} C_DIS
LIN {X 0.029,Y -141.470,Z 1507.149,A 0.000,B 0.000,C 90.000,E1 206.873} C_DIS
LIN {X 0.019,Y -139.378,Z 1507.113,A 0.000,B 0.000,C 90.000,E1 200.375} C_DIS
LIN {X 0.009,Y -138.830,Z 1507.098,A 0.000,B 0.000,C 90.000,E1 197.583} C_DIS
LIN {X -0.063,Y -138.353,Z 1507.056,A 0.000,B 0.000,C 90.000,E1 190.141} C_DIS
LIN {X -0.068,Y -139.527,Z 1507.004,A 0.000,B 0.000,C 90.000,E1 180.802} C_DIS
LIN {X 0.024,Y -141.200,Z 1506.973,A 0.000,B 0.000,C 90.000,E1 175.179} C_DIS
LIN {X -0.016,Y -142.576,Z 1506.958,A 0.000,B 0.000,C 90.000,E1 172.413} C_DIS
LIN {X 0.080,Y -144.868,Z 1506.932,A 0.000,B 0.000,C 90.000,E1 167.757} C_DIS
LIN {X 0.034,Y -147.494,Z 1506.912,A 0.000,B 0.000,C 90.000,E1 164.102} C_DIS
LIN {X -0.032,Y -150.083,Z 1506.891,A 0.000,B 0.000,C 90.000,E1 160.477} C_DIS
LIN {X -0.018,Y -153.436,Z 1506.871,A 0.000,B 0.000,C 90.000,E1 156.847} C_DIS
LIN {X -0.031,Y -156.855,Z 1506.851,A 0.000,B 0.000,C 90.000,E1 153.256} C_DIS
LIN {X 0.040,Y -160.938,Z 1506.832,A 0.000,B 0.000,C 90.000,E1 149.665} C_DIS
LIN {X -0.016,Y -163.062,Z 1506.822,A 0.000,B 0.000,C 90.000,E1 147.916} C_DIS
LIN {X -0.012,Y -167.458,Z 1506.802,A 0.000,B 0.000,C 90.000,E1 144.402} C_DIS
LIN {X 0.031,Y -171.294,Z 1506.788,A 0.000,B 0.000,C 90.000,E1 141.778} C_DIS
LIN {X 0.067,Y -176.190,Z 1506.769,A 0.000,B 0.000,C 90.000,E1 138.324} C_DIS
LIN {X -0.068,Y -180.464,Z 1506.754,A 0.000,B 0.000,C 90.000,E1 135.810} C_DIS
LIN {X -0.094,Y -185.869,Z 1506.736,A 0.000,B 0.000,C 90.000,E1 132.447} C_DIS
LIN {X -0.041,Y -190.494,Z 1506.722,A 0.000,B 0.000,C 90.000,E1 129.930} C_DIS
LIN {X -0.020,Y -196.245,Z 1506.703,A 0.000,B 0.000,C 90.000,E1 126.629} C_DIS
LIN {X -0.008,Y -201.376,Z 1506.689,A 0.000,B 0.000,C 90.000,E1 123.992} C_DIS
LIN {X 0.019,Y -201.992,Z 1506.687,A 0.000,B 0.000,C 90.000,E1 123.627} C_DIS
LIN {X -0.013,Y -316.035,Z 1506.687,A 0.000,B 0.000,C 90.000,E1 123.627} C_DIS
LIN {X 0.002,Y -322.451,Z 1506.685,A 0.000,B 0.000,C 90.000,E1 123.372} C_DIS
LIN {X 0.137,Y -325.435,Z 1506.684,A 0.000,B 0.000,C 90.000,E1 123.086} C_DIS
LIN {X -0.103,Y -329.122,Z 1506.681,A 0.000,B 0.000,C 90.000,E1 122.625} C_DIS
LIN {X -0.001,Y -330.741,Z 1506.679,A 0.000,B 0.000,C 90.000,E1 122.291} C_DIS
LIN {X -0.038,Y -345.705,Z 1506.659,A 0.000,B 0.000,C 90.000,E1 118.565} C_DIS
LIN {X -0.154,Y -358.470,Z 1506.643,A 0.000,B 0.000,C 90.000,E1 115.848} C_DIS
LIN {X 0.103,Y -372.749,Z 1506.629,A 0.000,B 0.000,C 90.000,E1 113.131} C_DIS
LIN {X 0.196,Y -386.817,Z 1506.616,A 0.000,B 0.000,C 90.000,E1 110.791} C_DIS
LIN {X 0.008,Y -402.278,Z 1506.603,A 0.000,B 0.000,C 90.000,E1 108.544} C_DIS
LIN {X 0.068,Y -419.243,Z 1506.591,A 0.000,B 0.000,C 90.000,E1 106.315} C_DIS
LIN {X -0.109,Y -437.826,Z 1506.579,A 0.000,B 0.000,C 90.000,E1 104.175} C_DIS
LIN {X -0.124,Y -457.682,Z 1506.567,A 0.000,B 0.000,C 90.000,E1 102.119} C_DIS
LIN {X 0.117,Y -478.116,Z 1506.557,A 0.000,B 0.000,C 90.000,E1 100.197} C_DIS
LIN {X 0.091,Y -491.015,Z 1506.551,A 0.000,B 0.000,C 90.000,E1 99.095} C_DIS
LIN {X 0.192,Y -492.971,Z 1506.549,A 0.000,B 0.000,C 90.000,E1 98.859} C_DIS
LIN {X -0.196,Y -494.465,Z 1506.548,A 0.000,B 0.000,C 90.000,E1 98.681} C_DIS
LIN {X 0.131,Y -495.706,Z 1506.547,A 0.000,B 0.000,C 90.000,E1 98.398} C_DIS
LIN {X 0.042,Y -496.610,Z 1506.545,A 0.000,B 0.000,C 90.000,E1 98.163} C_DIS
LIN {X -0.194,Y -497.568,Z 1506.543,A 0.000,B 0.000,C 90.000,E1 97.701} C_DIS
LIN {X 0.070,Y -497.515,Z 1506.540,A 0.000,B 0.000,C 90.000,E1 97.182} C_DIS
LIN {X -0.153,Y -496.448,Z 1506.537,A 0.000,B 0.000,C 90.000,E1 96.720} C_DIS
LIN {X 0.256,Y -495.483,Z 1506.536,A 0.000,B 0.000,C 90.000,E1 96.429} C_DIS
LIN {X 0.116,Y -494.172,Z 1506.535,A 0.000,B 0.000,C 90.000,E1 96.201} C_DIS
LIN {X -0.153,Y -484.333,Z 1506.526,A 0.000,B 0.000,C 90.000,E1 94.759} C_DIS
LIN {X -0.171,Y -475.263,Z 1506.518,A 0.000,B 0.000,C 90.000,E1 93.269} C_DIS
LIN {X -0.136,Y -467.276,Z 1506.511,A 0.000,B 0.000,C 90.000,E1 92.007} C_DIS
LIN {X 0.024,Y -457.079,Z 1506.503,A 0.000,B 0.000,C 90.000,E1 90.458} C_DIS
LIN {X -0.005,Y -446.571,Z 1506.494,A 0.000,B 0.000,C 90.000,E1 88.912} C_DIS
LIN {X 0.067,Y -437.660,Z 1506.487,A 0.000,B 0.000,C 90.000,E1 87.593} C_DIS
LIN {X 0.004,Y -423.091,Z 1506.475,A 0.000,B 0.000,C 90.000,E1 85.469} C_DIS
LIN {X -0.031,Y -410.409,Z 1506.464,A 0.000,B 0.000,C 90.000,E1 83.571} C_DIS
LIN {X -0.194,Y -395.912,Z 1506.452,A 0.000,B 0.000,C 90.000,E1 81.376} C_DIS
LIN {X -0.078,Y -374.960,Z 1506.433,A 0.000,B 0.000,C 90.000,E1 77.937} C_DIS
LIN {X 0.018,Y -360.230,Z 1506.418,A 0.000,B 0.000,C 90.000,E1 75.283} C_DIS
LIN {X -0.052,Y -348.967,Z 1506.407,A 0.000,B 0.000,C 90.000,E1 73.196} C_DIS
LIN {X 0.067,Y -336.200,Z 1506.393,A 0.000,B 0.000,C 90.000,E1 70.732} C_DIS
LIN {X -0.059,Y -319.269,Z 1506.374,A 0.000,B 0.000,C 90.000,E1 67.305} C_DIS
LIN {X -0.056,Y -306.233,Z 1506.358,A 0.000,B 0.000,C 90.000,E1 64.409} C_DIS
LIN {X 0.001,Y -292.484,Z 1506.339,A 0.000,B 0.000,C 90.000,E1 61.101} C_DIS
LIN {X -0.011,Y -281.986,Z 1506.324,A 0.000,B 0.000,C 90.000,E1 58.408} C_DIS
LIN {X 0.003,Y -270.587,Z 1506.307,A 0.000,B 0.000,C 90.000,E1 55.308} C_DIS
LIN {X 0.108,Y -260.804,Z 1506.292,A 0.000,B 0.000,C 90.000,E1 52.477} C_DIS
LIN {X -0.098,Y -250.263,Z 1506.274,A 0.000,B 0.000,C 90.000,E1 49.299} C_DIS
LIN {X 0.071,Y -240.462,Z 1506.255,A 0.000,B 0.000,C 90.000,E1 45.972} C_DIS
LIN {X 0.015,Y -232.439,Z 1506.239,A 0.000,B 0.000,C 90.000,E1 43.014} C_DIS
LIN {X -0.054,Y -225.243,Z 1506.222,A 0.000,B 0.000,C 90.000,E1 40.011} C_DIS
LIN {X -0.069,Y -218.749,Z 1506.205,A 0.000,B 0.000,C 90.000,E1 36.950} C_DIS
LIN {X -0.029,Y -212.889,Z 1506.188,A 0.000,B 0.000,C 90.000,E1 33.833} C_DIS
LIN {X 0.054,Y -206.334,Z 1506.166,A 0.000,B 0.000,C 90.000,E1 29.873} C_DIS
LIN {X -0.012,Y -200.673,Z 1506.144,A 0.000,B 0.000,C 90.000,E1 25.899} C_DIS
LIN {X 0.038,Y -195.803,Z 1506.121,A 0.000,B 0.000,C 90.000,E1 21.844} C_DIS
LIN {X 0.027,Y -191.763,Z 1506.099,A 0.000,B 0.000,C 90.000,E1 17.764} C_DIS
LIN {X -0.003,Y -187.816,Z 1506.071,A 0.000,B 0.000,C 90.000,E1 12.827} C_DIS
LIN {X 0.002,Y -184.678,Z 1506.039,A 0.000,B 0.000,C 90.000,E1 7.004} C_DIS
LIN {X -0.033,Y -182.856,Z 1505.997,A 0.000,B 0.000,C 90.000,E1 359.542} C_DIS
LIN {X 0.090,Y -183.466,Z 1505.955,A 0.000,B 0.000,C 90.000,E1 351.951} C_DIS
LIN {X 0.009,Y -186.063,Z 1505.918,A 0.000,B 0.000,C 90.000,E1 345.283} C_DIS
LIN {X -0.001,Y -189.438,Z 1505.891,A 0.000,B 0.000,C 90.000,E1 340.296} C_DIS
LIN {X -0.028,Y -193.194,Z 1505.868,A 0.000,B 0.000,C 90.000,E1 336.177} C_DIS
LIN {X -0.087,Y -197.805,Z 1505.845,A 0.000,B 0.000,C 90.000,E1 332.103} C_DIS
LIN {X -0.046,Y -203.400,Z 1505.822,A 0.000,B 0.000,C 90.000,E1 328.043} C_DIS
LIN {X 0.049,Y -208.704,Z 1505.805,A 0.000,B 0.000,C 90.000,E1 324.815} C_DIS
LIN {X 0.008,Y -214.758,Z 1505.787,A 0.000,B 0.000,C 90.000,E1 321.662} C_DIS
LIN {X 0.052,Y -221.654,Z 1505.770,A 0.000,B 0.000,C 90.000,E1 318.528} C_DIS
LIN {X -0.079,Y -229.461,Z 1505.753,A 0.000,B 0.000,C 90.000,E1 315.486} C_DIS
LIN {X -0.001,Y -238.268,Z 1505.736,A 0.000,B 0.000,C 90.000,E1 312.447} C_DIS
LIN {X -0.001,Y -248.215,Z 1505.719,A 0.000,B 0.000,C 90.000,E1 309.483} C_DIS
LIN {X 0.052,Y -255.233,Z 1505.709,A 0.000,B 0.000,C 90.000,E1 307.649} C_DIS
LIN {X -0.096,Y -263.205,Z 1505.699,A 0.000,B 0.000,C 90.000,E1 305.884} C_DIS
LIN {X -0.115,Y -272.113,Z 1505.689,A 0.000,B 0.000,C 90.000,E1 304.119} C_DIS
LIN {X 0.079,Y -282.168,Z 1505.680,A 0.000,B 0.000,C 90.000,E1 302.339} C_DIS
LIN {X -0.116,Y -295.467,Z 1505.668,A 0.000,B 0.000,C 90.000,E1 300.335} C_DIS
LIN {X 0.155,Y -305.151,Z 1505.661,A 0.000,B 0.000,C 90.000,E1 298.949} C_DIS
LIN {X -0.002,Y -326.555,Z 1505.647,A 0.000,B 0.000,C 90.000,E1 296.411} C_DIS
LIN {X 0.081,Y -345.685,Z 1505.635,A 0.000,B 0.000,C 90.000,E1 294.335} C_DIS
LIN {X -0.044,Y -361.854,Z 1505.626,A 0.000,B 0.000,C 90.000,E1 292.695} C_DIS
LIN {X 0.003,Y -372.478,Z 1505.620,A 0.000,B 0.000,C 90.000,E1 291.589} C_DIS
LIN {X 0.082,Y -382.813,Z 1505.614,A 0.000,B 0.000,C 90.000,E1 290.482} C_DIS
LIN {X -0.106,Y -392.896,Z 1505.608,A 0.000,B 0.000,C 90.000,E1 289.396} C_DIS
LIN {X 0.097,Y -402.633,Z 1505.601,A 0.000,B 0.000,C 90.000,E1 288.236} C_DIS
LIN {X 0.059,Y -409.345,Z 1505.597,A 0.000,B 0.000,C 90.000,E1 287.402} C_DIS
LIN {X 0.092,Y -415.431,Z 1505.592,A 0.000,B 0.000,C 90.000,E1 286.567} C_DIS
LIN {X -0.227,Y -420.796,Z 1505.588,A 0.000,B 0.000,C 90.000,E1 285.788} C_DIS
LIN {X 0.168,Y -423.938,Z 1505.584,A 0.000,B 0.000,C 90.000,E1 285.190} C_DIS
LIN {X -0.078,Y -428.025,Z 1505.580,A 0.000,B 0.000,C 90.000,E1 284.411} C_DIS
LIN {X 0.014,Y -431.417,Z 1505.576,A 0.000,B 0.000,C 90.000,E1 283.592} C_DIS
LIN {X -0.043,Y -433.236,Z 1505.573,A 0.000,B 0.000,C 90.000,E1 283.063} C_DIS
LIN {X -0.092,Y -434.692,Z 1505.570,A 0.000,B 0.000,C 90.000,E1 282.535} C_DIS
LIN {X -0.131,Y -435.705,Z 1505.567,A 0.000,B 0.000,C 90.000,E1 282.007} C_DIS
LIN {X -0.162,Y -436.252,Z 1505.564,A 0.000,B 0.000,C 90.000,E1 281.478} C_DIS
LIN {X -0.189,Y -436.293,Z 1505.561,A 0.000,B 0.000,C 90.000,E1 280.950} C_DIS
LIN {X 0.214,Y -435.749,Z 1505.558,A 0.000,B 0.000,C 90.000,E1 280.366} C_DIS
LIN {X 0.113,Y -434.697,Z 1505.555,A 0.000,B 0.000,C 90.000,E1 279.849} C_DIS
LIN {X 0.083,Y -432.987,Z 1505.552,A 0.000,B 0.000,C 90.000,E1 279.321} C_DIS
LIN {X -0.024,Y -430.540,Z 1505.549,A 0.000,B 0.000,C 90.000,E1 278.803} C_DIS
LIN {X 0.160,Y -429.042,Z 1505.547,A 0.000,B 0.000,C 90.000,E1 278.511} C_DIS
LIN {X 0.033,Y -425.324,Z 1505.544,A 0.000,B 0.000,C 90.000,E1 277.992} C_DIS
LIN {X -0.054,Y -420.659,Z 1505.541,A 0.000,B 0.000,C 90.000,E1 277.466} C_DIS
LIN {X -0.122,Y -415.098,Z 1505.538,A 0.000,B 0.000,C 90.000,E1 276.947} C_DIS
LIN {X 0.107,Y -409.085,Z 1505.536,A 0.000,B 0.000,C 90.000,E1 276.429} C_DIS
LIN {X -0.095,Y -402.912,Z 1505.533,A 0.000,B 0.000,C 90.000,E1 276.030} C_DIS
LIN {X 0.094,Y -396.550,Z 1505.531,A 0.000,B 0.000,C 90.000,E1 275.625} C_DIS
LIN {X 0.141,Y -390.090,Z 1505.529,A 0.000,B 0.000,C 90.000,E1 275.277} C_DIS
LIN {X 0.149,Y -380.223,Z 1505.527,A 0.000,B 0.000,C 90.000,E1 274.821} C_DIS
LIN {X 0.055,Y -367.497,Z 1505.524,A 0.000,B 0.000,C 90.000,E1 274.302} C_DIS
LIN {X -0.170,Y -351.554,Z 1505.521,A 0.000,B 0.000,C 90.000,E1 273.726} C_DIS
LIN {X -0.164,Y -341.665,Z 1505.519,A 0.000,B 0.000,C 90.000,E1 273.383} C_DIS
LIN {X 0.101,Y -331.804,Z 1505.517,A 0.000,B 0.000,C 90.000,E1 273.037} C_DIS
LIN {X -0.155,Y -321.823,Z 1505.516,A 0.000,B 0.000,C 90.000,E1 272.808} C_DIS
LIN {X 0.092,Y -310.780,Z 1505.514,A 0.000,B 0.000,C 90.000,E1 272.522} C_DIS
LIN {X -0.041,Y -298.770,Z 1505.513,A 0.000,B 0.000,C 90.000,E1 272.350} C_DIS
LIN {X -0.027,Y -287.896,Z 1505.512,A 0.000,B 0.000,C 90.000,E1 272.236} C_DIS
LIN {X -0.063,Y -275.342,Z 1505.512,A 0.000,B 0.000,C 90.000,E1 272.178} C_DIS
LIN {X -0.075,Y -181.237,Z 1505.512,A 0.000,B 0.000,C 90.000,E1 272.178} C_DIS
LIN {X 0.028,Y -181.575,Z 1505.501,A 0.000,B 0.000,C 90.000,E1 270.115} C_DIS
LIN {X 0.016,Y -180.876,Z 1505.473,A 0.000,B 0.000,C 90.000,E1 265.065} C_DIS
LIN {X 0.072,Y -178.993,Z 1505.444,A 0.000,B 0.000,C 90.000,E1 259.982} C_DIS
LIN {X -0.009,Y -178.577,Z 1505.440,A 0.000,B 0.000,C 90.000,E1 259.162} C_DIS
LIN {X 0.053,Y -175.629,Z 1505.411,A 0.000,B 0.000,C 90.000,E1 254.047} C_DIS
LIN {X -0.049,Y -172.350,Z 1505.388,A 0.000,B 0.000,C 90.000,E1 249.806} C_DIS
LIN {X -0.094,Y -171.131,Z 1505.378,A 0.000,B 0.000,C 90.000,E1 248.103} C_DIS
LIN {X -0.049,Y -167.438,Z 1505.354,A 0.000,B 0.000,C 90.000,E1 243.768} C_DIS
LIN {X 0.034,Y -166.834,Z 1505.349,A 0.000,B 0.000,C 90.000,E1 242.871} C_DIS
LIN {X -0.049,Y -162.817,Z 1505.325,A 0.000,B 0.000,C 90.000,E1 238.535} C_DIS
LIN {X 0.014,Y -161.503,Z 1505.315,A 0.000,B 0.000,C 90.000,E1 236.755} C_DIS
LIN {X -0.032,Y -157.500,Z 1505.291,A 0.000,B 0.000,C 90.000,E1 232.351} C_DIS
LIN {X 0.002,Y -155.520,Z 1505.276,A 0.000,B 0.000,C 90.000,E1 229.666} C_DIS
LIN {X 0.051,Y -151.819,Z 1505.251,A 0.000,B 0.000,C 90.000,E1 225.162} C_DIS
LIN {X 0.064,Y -150.033,Z 1505.236,A 0.000,B 0.000,C 90.000,E1 222.447} C_DIS
LIN {X -0.022,Y -146.852,Z 1505.211,A 0.000,B 0.000,C 90.000,E1 217.935} C_DIS
LIN {X -0.004,Y -145.435,Z 1505.195,A 0.000,B 0.000,C 90.000,E1 215.185} C_DIS
LIN {X -0.008,Y -142.858,Z 1505.170,A 0.000,B 0.000,C 90.000,E1 210.590} C_DIS
LIN {X 0.044,Y -141.473,Z 1505.149,A 0.000,B 0.000,C 90.000,E1 206.873} C_DIS
LIN {X 0.035,Y -139.379,Z 1505.113,A 0.000,B 0.000,C 90.000,E1 200.375} C_DIS
LIN {X 0.025,Y -138.832,Z 1505.098,A 0.000,B 0.000,C 90.000,E1 197.583} C_DIS
LIN {X -0.047,Y -138.353,Z 1505.056,A 0.000,B 0.000,C 90.000,E1 190.141} C_DIS
LIN {X -0.052,Y -139.526,Z 1505.004,A 0.000,B 0.000,C 90.000,E1 180.802} C_DIS
LIN {X 0.040,Y -141.197,Z 1504.973,A 0.000,B 0.000,C 90.000,E1 175.179} C_DIS
LIN {X -0.001,Y -142.574,Z 1504.958,A 0.000,B 0.000,C 90.000,E1 172.413} C_DIS
LIN {X -0.045,Y -144.864,Z 1504.932,A 0.000,B 0.000,C 90.000,E1 167.813} C_DIS
LIN {X 0.051,Y -147.490,Z 1504.912,A 0.000,B 0.000,C 90.000,E1 164.102} C_DIS
LIN {X -0.016,Y -150.078,Z 1504.891,A 0.000,B 0.000,C 90.000,E1 160.477} C_DIS
LIN {X -0.002,Y -153.429,Z 1504.871,A 0.000,B 0.000,C 90.000,E1 156.847} C_DIS
LIN {X -0.014,Y -156.848,Z 1504.851,A 0.000,B 0.000,C 90.000,E1 153.256} C_DIS
LIN {X 0.057,Y -160.930,Z 1504.832,A 0.000,B 0.000,C 90.000,E1 149.665} C_DIS
LIN {X 0.001,Y -163.054,Z 1504.822,A 0.000,B 0.000,C 90.000,E1 147.916} C_DIS
LIN {X 0.006,Y -167.448,Z 1504.802,A 0.000,B 0.000,C 90.000,E1 144.402} C_DIS
LIN {X -0.086,Y -171.286,Z 1504.788,A 0.000,B 0.000,C 90.000,E1 141.823} C_DIS
LIN {X 0.085,Y -176.181,Z 1504.769,A 0.000,B 0.000,C 90.000,E1 138.324} C_DIS
LIN {X -0.049,Y -180.454,Z 1504.754,A 0.000,B 0.000,C 90.000,E1 135.810} C_DIS
LIN {X -0.075,Y -185.859,Z 1504.736,A 0.000,B 0.000,C 90.000,E1 132.447} C_DIS
LIN {X -0.021,Y -190.483,Z 1504.722,A 0.000,B 0.000,C 90.000,E1 129.930} C_DIS
LIN {X 0.000,Y -196.235,Z 1504.703,A 0.000,B 0.000,C 90.000,E1 126.629} C_DIS
LIN {X 0.013,Y -201.366,Z 1504.689,A 0.000,B 0.000,C 90.000,E1 123.992} C_DIS
LIN {X 0.014,Y -201.939,Z 1504.687,A 0.000,B 0.000,C 90.000,E1 123.658} C_DIS
LIN {X -0.026,Y -316.076,Z 1504.687,A 0.000,B 0.000,C 90.000,E1 123.658} C_DIS
LIN {X 0.092,Y -320.479,Z 1504.686,A 0.000,B 0.000,C 90.000,E1 123.499} C_DIS
LIN {X 0.033,Y -322.667,Z 1504.685,A 0.000,B 0.000,C 90.000,E1 123.372} C_DIS
LIN {X -0.048,Y -326.539,Z 1504.683,A 0.000,B 0.000,C 90.000,E1 123.007} C_DIS
LIN {X -0.097,Y -329.998,Z 1504.680,A 0.000,B 0.000,C 90.000,E1 122.467} C_DIS
LIN {X 0.114,Y -332.563,Z 1504.677,A 0.000,B 0.000,C 90.000,E1 121.799} C_DIS
LIN {X -0.036,Y -343.692,Z 1504.661,A 0.000,B 0.000,C 90.000,E1 119.027} C_DIS
LIN {X -0.047,Y -356.213,Z 1504.646,A 0.000,B 0.000,C 90.000,E1 116.283} C_DIS
LIN {X -0.004,Y -370.230,Z 1504.631,A 0.000,B 0.000,C 90.000,E1 113.590} C_DIS
LIN {X 0.175,Y -384.047,Z 1504.618,A 0.000,B 0.000,C 90.000,E1 111.227} C_DIS
LIN {X 0.053,Y -399.239,Z 1504.605,A 0.000,B 0.000,C 90.000,E1 108.960} C_DIS
LIN {X 0.035,Y -415.912,Z 1504.593,A 0.000,B 0.000,C 90.000,E1 106.732} C_DIS
LIN {X 0.197,Y -434.182,Z 1504.581,A 0.000,B 0.000,C 90.000,E1 104.537} C_DIS
LIN {X -0.024,Y -453.883,Z 1504.569,A 0.000,B 0.000,C 90.000,E1 102.479} C_DIS
LIN {X 0.067,Y -474.216,Z 1504.559,A 0.000,B 0.000,C 90.000,E1 100.546} C_DIS
LIN {X 0.054,Y -489.797,Z 1504.551,A 0.000,B 0.000,C 90.000,E1 99.208} C_DIS
LIN {X 0.217,Y -491.972,Z 1504.550,A 0.000,B 0.000,C 90.000,E1 98.973} C_DIS
LIN {X 0.082,Y -493.794,Z 1504.549,A 0.000,B 0.000,C 90.000,E1 98.746} C_DIS
LIN {X 0.022,Y -495.163,Z 1504.547,A 0.000,B 0.000,C 90.000,E1 98.511} C_DIS
LIN {X -0.224,Y -496.909,Z 1504.545,A 0.000,B 0.000,C 90.000,E1 98.049} C_DIS
LIN {X 0.032,Y -497.548,Z 1504.542,A 0.000,B 0.000,C 90.000,E1 97.530} C_DIS
LIN {X -0.195,Y -497.191,Z 1504.539,A 0.000,B 0.000,C 90.000,E1 97.068} C_DIS
LIN {X 0.076,Y -495.784,Z 1504.536,A 0.000,B 0.000,C 90.000,E1 96.549} C_DIS
LIN {X -0.008,Y -494.614,Z 1504.535,A 0.000,B 0.000,C 90.000,E1 96.315} C_DIS
LIN {X 0.056,Y -483.291,Z 1504.526,A 0.000,B 0.000,C 90.000,E1 94.588} C_DIS
LIN {X 0.045,Y -474.220,Z 1504.517,A 0.000,B 0.000,C 90.000,E1 93.094} C_DIS
LIN {X 0.038,Y -466.150,Z 1504.510,A 0.000,B 0.000,C 90.000,E1 91.835} C_DIS
LIN {X 0.175,Y -455.933,Z 1504.502,A 0.000,B 0.000,C 90.000,E1 90.286} C_DIS
LIN {X 0.124,Y -445.408,Z 1504.493,A 0.000,B 0.000,C 90.000,E1 88.740} C_DIS
LIN {X 0.175,Y -436.495,Z 1504.486,A 0.000,B 0.000,C 90.000,E1 87.421} C_DIS
LIN {X 0.079,Y -421.988,Z 1504.474,A 0.000,B 0.000,C 90.000,E1 85.298} C_DIS
LIN {X 0.062,Y -409.345,Z 1504.463,A 0.000,B 0.000,C 90.000,E1 83.394} C_DIS
LIN {X -0.120,Y -394.877,Z 1504.451,A 0.000,B 0.000,C 90.000,E1 81.197} C_DIS
LIN {X -0.032,Y -374.002,Z 1504.432,A 0.000,B 0.000,C 90.000,E1 77.757} C_DIS
LIN {X -0.020,Y -360.935,Z 1504.419,A 0.000,B 0.000,C 90.000,E1 75.408} C_DIS
LIN {X -0.075,Y -349.676,Z 1504.407,A 0.000,B 0.000,C 90.000,E1 73.323} C_DIS
LIN {X 0.056,Y -338.462,Z 1504.395,A 0.000,B 0.000,C 90.000,E1 71.167} C_DIS
LIN {X 0.086,Y -324.385,Z 1504.380,A 0.000,B 0.000,C 90.000,E1 68.358} C_DIS
LIN {X 0.092,Y -311.093,Z 1504.364,A 0.000,B 0.000,C 90.000,E1 65.485} C_DIS
LIN {X 0.001,Y -298.445,Z 1504.348,A 0.000,B 0.000,C 90.000,E1 62.564} C_DIS
LIN {X 0.111,Y -286.439,Z 1504.331,A 0.000,B 0.000,C 90.000,E1 59.537} C_DIS
LIN {X -0.006,Y -276.159,Z 1504.316,A 0.000,B 0.000,C 90.000,E1 56.834} C_DIS
LIN {X 0.002,Y -265.044,Z 1504.298,A 0.000,B 0.000,C 90.000,E1 53.703} C_DIS
LIN {X -0.050,Y -254.298,Z 1504.281,A 0.000,B 0.000,C 90.000,E1 50.517} C_DIS
LIN {X 0.058,Y -244.303,Z 1504.262,A 0.000,B 0.000,C 90.000,E1 47.229} C_DIS
LIN {X 0.028,Y -234.033,Z 1504.242,A 0.000,B 0.000,C 90.000,E1 43.542} C_DIS
LIN {X -0.005,Y -226.734,Z 1504.225,A 0.000,B 0.000,C 90.000,E1 40.539} C_DIS
LIN {X -0.023,Y -220.087,Z 1504.208,A 0.000,B 0.000,C 90.000,E1 37.488} C_DIS
LIN {X 0.092,Y -212.747,Z 1504.187,A 0.000,B 0.000,C 90.000,E1 33.579} C_DIS
LIN {X -0.006,Y -206.220,Z 1504.165,A 0.000,B 0.000,C 90.000,E1 29.667} C_DIS
LIN {X 0.014,Y -200.604,Z 1504.143,A 0.000,B 0.000,C 90.000,E1 25.668} C_DIS
LIN {X -0.037,Y -195.816,Z 1504.120,A 0.000,B 0.000,C 90.000,E1 21.642} C_DIS
LIN {X -0.117,Y -191.789,Z 1504.098,A 0.000,B 0.000,C 90.000,E1 17.583} C_DIS
LIN {X 0.039,Y -187.905,Z 1504.070,A 0.000,B 0.000,C 90.000,E1 12.591} C_DIS
LIN {X 0.019,Y -184.853,Z 1504.038,A 0.000,B 0.000,C 90.000,E1 6.777} C_DIS
LIN {X -0.033,Y -183.129,Z 1503.997,A 0.000,B 0.000,C 90.000,E1 359.542} C_DIS
LIN {X -0.077,Y -183.743,Z 1503.955,A 0.000,B 0.000,C 90.000,E1 352.008} C_DIS
LIN {X 0.037,Y -186.289,Z 1503.918,A 0.000,B 0.000,C 90.000,E1 345.283} C_DIS
LIN {X -0.028,Y -189.636,Z 1503.891,A 0.000,B 0.000,C 90.000,E1 340.315} C_DIS
LIN {X 0.014,Y -193.374,Z 1503.868,A 0.000,B 0.000,C 90.000,E1 336.177} C_DIS
LIN {X -0.036,Y -197.954,Z 1503.845,A 0.000,B 0.000,C 90.000,E1 332.103} C_DIS
LIN {X 0.009,Y -203.546,Z 1503.823,A 0.000,B 0.000,C 90.000,E1 328.043} C_DIS
LIN {X -0.011,Y -208.816,Z 1503.805,A 0.000,B 0.000,C 90.000,E1 324.848} C_DIS
LIN {X -0.061,Y -214.886,Z 1503.787,A 0.000,B 0.000,C 90.000,E1 321.698} C_DIS
LIN {X -0.024,Y -221.781,Z 1503.770,A 0.000,B 0.000,C 90.000,E1 318.566} C_DIS
LIN {X -0.002,Y -229.599,Z 1503.753,A 0.000,B 0.000,C 90.000,E1 315.486} C_DIS
LIN {X 0.082,Y -238.415,Z 1503.736,A 0.000,B 0.000,C 90.000,E1 312.447} C_DIS
LIN {X 0.089,Y -248.351,Z 1503.719,A 0.000,B 0.000,C 90.000,E1 309.483} C_DIS
LIN {X 0.014,Y -256.852,Z 1503.707,A 0.000,B 0.000,C 90.000,E1 307.317} C_DIS
LIN {X 0.054,Y -265.005,Z 1503.697,A 0.000,B 0.000,C 90.000,E1 305.518} C_DIS
LIN {X -0.093,Y -274.068,Z 1503.688,A 0.000,B 0.000,C 90.000,E1 303.785} C_DIS
LIN {X 0.144,Y -284.268,Z 1503.678,A 0.000,B 0.000,C 90.000,E1 302.005} C_DIS
LIN {X -0.007,Y -297.685,Z 1503.667,A 0.000,B 0.000,C 90.000,E1 300.001} C_DIS
LIN {X -0.120,Y -307.567,Z 1503.659,A 0.000,B 0.000,C 90.000,E1 298.693} C_DIS
LIN {X 0.007,Y -328.924,Z 1503.645,A 0.000,B 0.000,C 90.000,E1 296.155} C_DIS
LIN {X 0.124,Y -345.286,Z 1503.636,A 0.000,B 0.000,C 90.000,E1 294.387} C_DIS
LIN {X 0.115,Y -361.610,Z 1503.626,A 0.000,B 0.000,C 90.000,E1 292.717} C_DIS
LIN {X 0.069,Y -374.861,Z 1503.619,A 0.000,B 0.000,C 90.000,E1 291.354} C_DIS
LIN {X -0.164,Y -385.016,Z 1503.613,A 0.000,B 0.000,C 90.000,E1 290.301} C_DIS
LIN {X 0.034,Y -395.202,Z 1503.606,A 0.000,B 0.000,C 90.000,E1 289.141} C_DIS
LIN {X -0.070,Y -402.476,Z 1503.602,A 0.000,B 0.000,C 90.000,E1 288.308} C_DIS
LIN {X 0.014,Y -409.250,Z 1503.597,A 0.000,B 0.000,C 90.000,E1 287.457} C_DIS
LIN {X 0.044,Y -415.375,Z 1503.592,A 0.000,B 0.000,C 90.000,E1 286.622} C_DIS
LIN {X 0.126,Y -420.815,Z 1503.588,A 0.000,B 0.000,C 90.000,E1 285.788} C_DIS
LIN {X -0.143,Y -425.454,Z 1503.583,A 0.000,B 0.000,C 90.000,E1 285.009} C_DIS
LIN {X 0.030,Y -429.415,Z 1503.579,A 0.000,B 0.000,C 90.000,E1 284.175} C_DIS
LIN {X -0.042,Y -431.632,Z 1503.576,A 0.000,B 0.000,C 90.000,E1 283.647} C_DIS
LIN {X -0.098,Y -433.531,Z 1503.573,A 0.000,B 0.000,C 90.000,E1 283.119} C_DIS
LIN {X -0.148,Y -435.038,Z 1503.570,A 0.000,B 0.000,C 90.000,E1 282.591} C_DIS
LIN {X -0.186,Y -436.115,Z 1503.567,A 0.000,B 0.000,C 90.000,E1 282.063} C_DIS
LIN {X 0.212,Y -436.725,Z 1503.564,A 0.000,B 0.000,C 90.000,E1 281.478} C_DIS
LIN {X 0.188,Y -436.865,Z 1503.561,A 0.000,B 0.000,C 90.000,E1 280.950} C_DIS
LIN {X 0.086,Y -436.387,Z 1503.558,A 0.000,B 0.000,C 90.000,E1 280.433} C_DIS
LIN {X 0.065,Y -435.388,Z 1503.555,A 0.000,B 0.000,C 90.000,E1 279.905} C_DIS
LIN {X 0.039,Y -433.767,Z 1503.552,A 0.000,B 0.000,C 90.000,E1 279.378} C_DIS
LIN {X -0.064,Y -431.432,Z 1503.549,A 0.000,B 0.000,C 90.000,E1 278.859} C_DIS
LIN {X -0.178,Y -428.293,Z 1503.546,A 0.000,B 0.000,C 90.000,E1 278.341} C_DIS
LIN {X 0.175,Y -424.220,Z 1503.543,A 0.000,B 0.000,C 90.000,E1 277.757} C_DIS
LIN {X 0.026,Y -419.193,Z 1503.540,A 0.000,B 0.000,C 90.000,E1 277.239} C_DIS
LIN {X -0.017,Y -413.242,Z 1503.537,A 0.000,B 0.000,C 90.000,E1 276.720} C_DIS
LIN {X -0.001,Y -407.104,Z 1503.535,A 0.000,B 0.000,C 90.000,E1 276.258} C_DIS
LIN {X -0.037,Y -400.777,Z 1503.532,A 0.000,B 0.000,C 90.000,E1 275.853} C_DIS
LIN {X -0.150,Y -394.419,Z 1503.531,A 0.000,B 0.000,C 90.000,E1 275.511} C_DIS
LIN {X 0.042,Y -388.147,Z 1503.529,A 0.000,B 0.000,C 90.000,E1 275.163} C_DIS
LIN {X 0.068,Y -375.130,Z 1503.526,A 0.000,B 0.000,C 90.000,E1 274.588} C_DIS
LIN {X 0.061,Y -362.423,Z 1503.523,A 0.000,B 0.000,C 90.000,E1 274.073} C_DIS
LIN {X -0.045,Y -346.396,Z 1503.519,A 0.000,B 0.000,C 90.000,E1 273.498} C_DIS
LIN {X 0.041,Y -336.126,Z 1503.518,A 0.000,B 0.000,C 90.000,E1 273.154} C_DIS
LIN {X -0.074,Y -322.851,Z 1503.516,A 0.000,B 0.000,C 90.000,E1 272.808} C_DIS
LIN {X -0.124,Y -312.160,Z 1503.514,A 0.000,B 0.000,C 90.000,E1 272.579} C_DIS
LIN {X 0.031,Y -300.327,Z 1503.513,A 0.000,B 0.000,C 90.000,E1 272.350} C_DIS
LIN {X -0.086,Y -286.776,Z 1503.512,A 0.000,B 0.000,C 90.000,E1 272.236} C_DIS
LIN {X -0.025,Y -277.737,Z 1503.512,A 0.000,B 0.000,C 90.000,E1 272.178} C_DIS
LIN {X -0.052,Y -181.236,Z 1503.512,A 0.000,B 0.000,C 90.000,E1 272.178} C_DIS
LIN {X 0.050,Y -181.575,Z 1503.501,A 0.000,B 0.000,C 90.000,E1 270.115} C_DIS
LIN {X 0.038,Y -180.877,Z 1503.473,A 0.000,B 0.000,C 90.000,E1 265.065} C_DIS
LIN {X -0.082,Y -178.996,Z 1503.444,A 0.000,B 0.000,C 90.000,E1 260.038} C_DIS
LIN {X 0.012,Y -178.582,Z 1503.440,A 0.000,B 0.000,C 90.000,E1 259.162} C_DIS
LIN {X -0.094,Y -175.635,Z 1503.411,A 0.000,B 0.000,C 90.000,E1 254.102} C_DIS
LIN {X -0.028,Y -172.354,Z 1503.388,A 0.000,B 0.000,C 90.000,E1 249.806} C_DIS
LIN {X -0.073,Y -171.138,Z 1503.378,A 0.000,B 0.000,C 90.000,E1 248.103} C_DIS
LIN {X -0.028,Y -167.443,Z 1503.354,A 0.000,B 0.000,C 90.000,E1 243.768} C_DIS
LIN {X 0.054,Y -166.839,Z 1503.349,A 0.000,B 0.000,C 90.000,E1 242.871} C_DIS
LIN {X -0.029,Y -162.822,Z 1503.325,A 0.000,B 0.000,C 90.000,E1 238.535} C_DIS
LIN {X 0.035,Y -161.508,Z 1503.315,A 0.000,B 0.000,C 90.000,E1 236.755} C_DIS
LIN {X -0.012,Y -157.506,Z 1503.291,A 0.000,B 0.000,C 90.000,E1 232.351} C_DIS
LIN {X 0.022,Y -155.527,Z 1503.276,A 0.000,B 0.000,C 90.000,E1 229.666} C_DIS
LIN {X 0.071,Y -151.825,Z 1503.251,A 0.000,B 0.000,C 90.000,E1 225.162} C_DIS
LIN {X 0.084,Y -150.040,Z 1503.236,A 0.000,B 0.000,C 90.000,E1 222.447} C_DIS
LIN {X -0.003,Y -146.856,Z 1503.211,A 0.000,B 0.000,C 90.000,E1 217.935} C_DIS
LIN {X 0.016,Y -145.440,Z 1503.196,A 0.000,B 0.000,C 90.000,E1 215.185} C_DIS
LIN {X 0.011,Y -142.861,Z 1503.170,A 0.000,B 0.000,C 90.000,E1 210.590} C_DIS
LIN {X 0.063,Y -141.477,Z 1503.149,A 0.000,B 0.000,C 90.000,E1 206.873} C_DIS
LIN {X -0.077,Y -139.380,Z 1503.113,A 0.000,B 0.000,C 90.000,E1 200.429} C_DIS
LIN {X 0.044,Y -138.834,Z 1503.098,A 0.000,B 0.000,C 90.000,E1 197.583} C_DIS
LIN {X -0.028,Y -138.353,Z 1503.056,A 0.000,B 0.000,C 90.000,E1 190.141} C_DIS
LIN {X -0.033,Y -139.525,Z 1503.004,A 0.000,B 0.000,C 90.000,E1 180.802} C_DIS
LIN {X 0.059,Y -141.195,Z 1502.973,A 0.000,B 0.000,C 90.000,E1 175.179} C_DIS
LIN {X 0.018,Y -142.571,Z 1502.958,A 0.000,B 0.000,C 90.000,E1 172.413} C_DIS
LIN {X -0.027,Y -144.859,Z 1502.932,A 0.000,B 0.000,C 90.000,E1 167.813} C_DIS
LIN {X -0.072,Y -147.485,Z 1502.912,A 0.000,B 0.000,C 90.000,E1 164.157} C_DIS
LIN {X -0.046,Y -150.072,Z 1502.892,A 0.000,B 0.000,C 90.000,E1 160.496} C_DIS
LIN {X -0.042,Y -153.421,Z 1502.871,A 0.000,B 0.000,C 90.000,E1 156.869} C_DIS
LIN {X 0.006,Y -156.842,Z 1502.851,A 0.000,B 0.000,C 90.000,E1 153.256} C_DIS
LIN {X 0.078,Y -160.922,Z 1502.832,A 0.000,B 0.000,C 90.000,E1 149.665} C_DIS
LIN {X 0.022,Y -163.046,Z 1502.822,A 0.000,B 0.000,C 90.000,E1 147.916} C_DIS
LIN {X 0.027,Y -167.440,Z 1502.802,A 0.000,B 0.000,C 90.000,E1 144.402} C_DIS
LIN {X -0.064,Y -171.277,Z 1502.788,A 0.000,B 0.000,C 90.000,E1 141.823} C_DIS
LIN {X -0.026,Y -176.170,Z 1502.769,A 0.000,B 0.000,C 90.000,E1 138.366} C_DIS
LIN {X -0.028,Y -180.442,Z 1502.754,A 0.000,B 0.000,C 90.000,E1 135.810} C_DIS
LIN {X -0.053,Y -185.847,Z 1502.736,A 0.000,B 0.000,C 90.000,E1 132.447} C_DIS
LIN {X 0.001,Y -190.470,Z 1502.722,A 0.000,B 0.000,C 90.000,E1 129.930} C_DIS
LIN {X -0.095,Y -196.222,Z 1502.703,A 0.000,B 0.000,C 90.000,E1 126.664} C_DIS
LIN {X 0.037,Y -201.354,Z 1502.689,A 0.000,B 0.000,C 90.000,E1 123.992} C_DIS
LIN {X -0.038,Y -201.882,Z 1502.687,A 0.000,B 0.000,C 90.000,E1 123.706} C_DIS
LIN {X -0.107,Y -315.834,Z 1502.687,A 0.000,B 0.000,C 90.000,E1 123.706} C_DIS
LIN {X 0.014,Y -317.352,Z 1502.687,A 0.000,B 0.000,C 90.000,E1 123.658} C_DIS
LIN {X 0.071,Y -322.862,Z 1502.685,A 0.000,B 0.000,C 90.000,E1 123.372} C_DIS
LIN {X -0.058,Y -326.025,Z 1502.684,A 0.000,B 0.000,C 90.000,E1 123.086} C_DIS
LIN {X -0.093,Y -329.617,Z 1502.681,A 0.000,B 0.000,C 90.000,E1 122.546} C_DIS
LIN {X 0.011,Y -331.065,Z 1502.679,A 0.000,B 0.000,C 90.000,E1 122.212} C_DIS
LIN {X 0.128,Y -343.340,Z 1502.662,A 0.000,B 0.000,C 90.000,E1 119.077} C_DIS
LIN {X -0.052,Y -355.821,Z 1502.646,A 0.000,B 0.000,C 90.000,E1 116.360} C_DIS
LIN {X 0.135,Y -369.794,Z 1502.631,A 0.000,B 0.000,C 90.000,E1 113.643} C_DIS
LIN {X -0.055,Y -383.569,Z 1502.619,A 0.000,B 0.000,C 90.000,E1 111.334} C_DIS
LIN {X 0.039,Y -398.716,Z 1502.606,A 0.000,B 0.000,C 90.000,E1 109.033} C_DIS
LIN {X 0.018,Y -415.340,Z 1502.593,A 0.000,B 0.000,C 90.000,E1 106.804} C_DIS
LIN {X -0.135,Y -433.558,Z 1502.581,A 0.000,B 0.000,C 90.000,E1 104.647} C_DIS
LIN {X 0.030,Y -453.227,Z 1502.570,A 0.000,B 0.000,C 90.000,E1 102.535} C_DIS
LIN {X 0.077,Y -473.544,Z 1502.559,A 0.000,B 0.000,C 90.000,E1 100.602} C_DIS
LIN {X 0.032,Y -489.118,Z 1502.552,A 0.000,B 0.000,C 90.000,E1 99.265} C_DIS
LIN {X 0.190,Y -491.443,Z 1502.550,A 0.000,B 0.000,C 90.000,E1 99.029} C_DIS
LIN {X 0.131,Y -493.310,Z 1502.549,A 0.000,B 0.000,C 90.000,E1 98.803} C_DIS
LIN {X 0.147,Y -494.726,Z 1502.548,A 0.000,B 0.000,C 90.000,E1 98.568} C_DIS
LIN {X -0.101,Y -496.639,Z 1502.545,A 0.000,B 0.000,C 90.000,E1 98.106} C_DIS
LIN {X 0.151,Y -497.414,Z 1502.542,A 0.000,B 0.000,C 90.000,E1 97.587} C_DIS
LIN {X -0.077,Y -497.188,Z 1502.540,A 0.000,B 0.000,C 90.000,E1 97.125} C_DIS
LIN {X 0.193,Y -495.929,Z 1502.537,A 0.000,B 0.000,C 90.000,E1 96.606} C_DIS
LIN {X 0.107,Y -494.850,Z 1502.536,A 0.000,B 0.000,C 90.000,E1 96.372} C_DIS
LIN {X -0.032,Y -493.398,Z 1502.534,A 0.000,B 0.000,C 90.000,E1 96.144} C_DIS
LIN {X -0.194,Y -485.124,Z 1502.527,A 0.000,B 0.000,C 90.000,E1 94.935} C_DIS
LIN {X 0.138,Y -474.520,Z 1502.518,A 0.000,B 0.000,C 90.000,E1 93.154} C_DIS
LIN {X 0.158,Y -466.506,Z 1502.511,A 0.000,B 0.000,C 90.000,E1 91.892} C_DIS
LIN {X -0.157,Y -456.307,Z 1502.502,A 0.000,B 0.000,C 90.000,E1 90.401} C_DIS
LIN {X -0.195,Y -445.812,Z 1502.494,A 0.000,B 0.000,C 90.000,E1 88.854} C_DIS
LIN {X 0.034,Y -435.103,Z 1502.485,A 0.000,B 0.000,C 90.000,E1 87.249} C_DIS
LIN {X -0.057,Y -420.677,Z 1502.473,A 0.000,B 0.000,C 90.000,E1 85.122} C_DIS
LIN {X 0.160,Y -409.873,Z 1502.464,A 0.000,B 0.000,C 90.000,E1 83.457} C_DIS
LIN {X 0.034,Y -395.423,Z 1502.451,A 0.000,B 0.000,C 90.000,E1 81.254} C_DIS
LIN {X 0.057,Y -374.514,Z 1502.432,A 0.000,B 0.000,C 90.000,E1 77.825} C_DIS
LIN {X 0.188,Y -363.071,Z 1502.421,A 0.000,B 0.000,C 90.000,E1 75.755} C_DIS
LIN {X 0.074,Y -351.805,Z 1502.409,A 0.000,B 0.000,C 90.000,E1 73.685} C_DIS
LIN {X -0.074,Y -340.556,Z 1502.398,A 0.000,B 0.000,C 90.000,E1 71.583} C_DIS
LIN {X 0.077,Y -329.458,Z 1502.386,A 0.000,B 0.000,C 90.000,E1 69.390} C_DIS
LIN {X 0.042,Y -314.407,Z 1502.368,A 0.000,B 0.000,C 90.000,E1 66.230} C_DIS
LIN {X -0.083,Y -301.605,Z 1502.352,A 0.000,B 0.000,C 90.000,E1 63.332} C_DIS
LIN {X -0.031,Y -288.151,Z 1502.333,A 0.000,B 0.000,C 90.000,E1 59.999} C_DIS
LIN {X 0.134,Y -277.841,Z 1502.318,A 0.000,B 0.000,C 90.000,E1 57.248} C_DIS
LIN {X 0.106,Y -267.895,Z 1502.303,A 0.000,B 0.000,C 90.000,E1 54.482} C_DIS
LIN {X -0.072,Y -258.284,Z 1502.287,A 0.000,B 0.000,C 90.000,E1 51.698} C_DIS
LIN {X 0.154,Y -249.172,Z 1502.271,A 0.000,B 0.000,C 90.000,E1 48.771} C_DIS
LIN {X -0.066,Y -238.561,Z 1502.251,A 0.000,B 0.000,C 90.000,E1 45.162} C_DIS
LIN {X 0.005,Y -230.793,Z 1502.234,A 0.000,B 0.000,C 90.000,E1 42.162} C_DIS
LIN {X -0.056,Y -222.173,Z 1502.213,A 0.000,B 0.000,C 90.000,E1 38.382} C_DIS
LIN {X 0.079,Y -214.599,Z 1502.192,A 0.000,B 0.000,C 90.000,E1 34.485} C_DIS
LIN {X -0.027,Y -207.901,Z 1502.170,A 0.000,B 0.000,C 90.000,E1 30.590} C_DIS
LIN {X -0.043,Y -202.058,Z 1502.148,A 0.000,B 0.000,C 90.000,E1 26.616} C_DIS
LIN {X -0.047,Y -197.096,Z 1502.125,A 0.000,B 0.000,C 90.000,E1 22.589} C_DIS
LIN {X 0.050,Y -192.882,Z 1502.103,A 0.000,B 0.000,C 90.000,E1 18.489} C_DIS
LIN {X -0.070,Y -188.810,Z 1502.075,A 0.000,B 0.000,C 90.000,E1 13.592} C_DIS
LIN {X 0.013,Y -185.511,Z 1502.043,A 0.000,B 0.000,C 90.000,E1 7.757} C_DIS
LIN {X -0.035,Y -183.568,Z 1502.006,A 0.000,B 0.000,C 90.000,E1 1.088} C_DIS
LIN {X -0.067,Y -183.667,Z 1501.965,A 0.000,B 0.000,C 90.000,E1 353.685} C_DIS
LIN {X 0.063,Y -186.073,Z 1501.923,A 0.000,B 0.000,C 90.000,E1 346.117} C_DIS
LIN {X -0.007,Y -189.198,Z 1501.895,A 0.000,B 0.000,C 90.000,E1 341.148} C_DIS
LIN {X -0.112,Y -192.743,Z 1501.872,A 0.000,B 0.000,C 90.000,E1 337.050} C_DIS
LIN {X -0.005,Y -197.133,Z 1501.850,A 0.000,B 0.000,C 90.000,E1 332.922} C_DIS
LIN {X -0.009,Y -202.480,Z 1501.827,A 0.000,B 0.000,C 90.000,E1 328.869} C_DIS
LIN {X -0.057,Y -207.554,Z 1501.809,A 0.000,B 0.000,C 90.000,E1 325.674} C_DIS
LIN {X 0.036,Y -213.405,Z 1501.792,A 0.000,B 0.000,C 90.000,E1 322.477} C_DIS
LIN {X -0.098,Y -220.106,Z 1501.774,A 0.000,B 0.000,C 90.000,E1 319.380} C_DIS
LIN {X -0.115,Y -227.683,Z 1501.757,A 0.000,B 0.000,C 90.000,E1 316.296} C_DIS
LIN {X 0.078,Y -236.260,Z 1501.740,A 0.000,B 0.000,C 90.000,E1 313.218} C_DIS
LIN {X 0.024,Y -247.173,Z 1501.722,A 0.000,B 0.000,C 90.000,E1 309.886} C_DIS
LIN {X -0.115,Y -255.480,Z 1501.709,A 0.000,B 0.000,C 90.000,E1 307.729} C_DIS
LIN {X 0.105,Y -263.410,Z 1501.699,A 0.000,B 0.000,C 90.000,E1 305.884} C_DIS
LIN {X 0.095,Y -272.238,Z 1501.690,A 0.000,B 0.000,C 90.000,E1 304.119} C_DIS
LIN {X -0.090,Y -282.128,Z 1501.680,A 0.000,B 0.000,C 90.000,E1 302.418} C_DIS
LIN {X 0.114,Y -295.281,Z 1501.669,A 0.000,B 0.000,C 90.000,E1 300.335} C_DIS
LIN {X -0.011,Y -304.854,Z 1501.661,A 0.000,B 0.000,C 90.000,E1 299.027} C_DIS
LIN {X -0.103,Y -323.457,Z 1501.649,A 0.000,B 0.000,C 90.000,E1 296.796} C_DIS
LIN {X -0.110,Y -345.095,Z 1501.636,A 0.000,B 0.000,C 90.000,E1 294.463} C_DIS
LIN {X 0.034,Y -361.440,Z 1501.627,A 0.000,B 0.000,C 90.000,E1 292.770} C_DIS
LIN {X -0.034,Y -374.726,Z 1501.619,A 0.000,B 0.000,C 90.000,E1 291.408} C_DIS
LIN {X -0.055,Y -385.067,Z 1501.613,A 0.000,B 0.000,C 90.000,E1 290.301} C_DIS
LIN {X 0.124,Y -395.320,Z 1501.606,A 0.000,B 0.000,C 90.000,E1 289.141} C_DIS
LIN {X 0.024,Y -402.608,Z 1501.602,A 0.000,B 0.000,C 90.000,E1 288.308} C_DIS
LIN {X 0.111,Y -409.386,Z 1501.597,A 0.000,B 0.000,C 90.000,E1 287.457} C_DIS
LIN {X 0.032,Y -413.609,Z 1501.594,A 0.000,B 0.000,C 90.000,E1 286.913} C_DIS
LIN {X 0.102,Y -419.292,Z 1501.589,A 0.000,B 0.000,C 90.000,E1 286.079} C_DIS
LIN {X 0.220,Y -424.243,Z 1501.585,A 0.000,B 0.000,C 90.000,E1 285.245} C_DIS
LIN {X -0.133,Y -428.471,Z 1501.580,A 0.000,B 0.000,C 90.000,E1 284.481} C_DIS
LIN {X 0.070,Y -431.989,Z 1501.576,A 0.000,B 0.000,C 90.000,E1 283.647} C_DIS
LIN {X 0.016,Y -433.901,Z 1501.573,A 0.000,B 0.000,C 90.000,E1 283.119} C_DIS
LIN {X -0.031,Y -435.448,Z 1501.570,A 0.000,B 0.000,C 90.000,E1 282.591} C_DIS
LIN {X -0.067,Y -436.576,Z 1501.567,A 0.000,B 0.000,C 90.000,E1 282.063} C_DIS
LIN {X -0.094,Y -437.225,Z 1501.564,A 0.000,B 0.000,C 90.000,E1 281.535} C_DIS
LIN {X -0.117,Y -437.389,Z 1501.561,A 0.000,B 0.000,C 90.000,E1 281.007} C_DIS
LIN {X -0.217,Y -436.954,Z 1501.558,A 0.000,B 0.000,C 90.000,E1 280.489} C_DIS
LIN {X 0.196,Y -436.012,Z 1501.555,A 0.000,B 0.000,C 90.000,E1 279.905} C_DIS
LIN {X 0.171,Y -434.395,Z 1501.552,A 0.000,B 0.000,C 90.000,E1 279.378} C_DIS
LIN {X 0.072,Y -432.133,Z 1501.549,A 0.000,B 0.000,C 90.000,E1 278.859} C_DIS
LIN {X -0.040,Y -429.045,Z 1501.546,A 0.000,B 0.000,C 90.000,E1 278.341} C_DIS
LIN {X -0.104,Y -425.074,Z 1501.543,A 0.000,B 0.000,C 90.000,E1 277.814} C_DIS
LIN {X 0.171,Y -420.048,Z 1501.540,A 0.000,B 0.000,C 90.000,E1 277.239} C_DIS
LIN {X -0.040,Y -417.257,Z 1501.539,A 0.000,B 0.000,C 90.000,E1 277.004} C_DIS
LIN {X 0.145,Y -411.219,Z 1501.536,A 0.000,B 0.000,C 90.000,E1 276.486} C_DIS
LIN {X -0.126,Y -405.049,Z 1501.534,A 0.000,B 0.000,C 90.000,E1 276.087} C_DIS
LIN {X -0.021,Y -398.657,Z 1501.531,A 0.000,B 0.000,C 90.000,E1 275.682} C_DIS
LIN {X 0.004,Y -392.151,Z 1501.530,A 0.000,B 0.000,C 90.000,E1 275.334} C_DIS
LIN {X 0.004,Y -382.324,Z 1501.527,A 0.000,B 0.000,C 90.000,E1 274.878} C_DIS
LIN {X -0.115,Y -369.616,Z 1501.524,A 0.000,B 0.000,C 90.000,E1 274.359} C_DIS
LIN {X 0.022,Y -356.796,Z 1501.521,A 0.000,B 0.000,C 90.000,E1 273.841} C_DIS
LIN {X -0.013,Y -343.892,Z 1501.519,A 0.000,B 0.000,C 90.000,E1 273.383} C_DIS
LIN {X -0.132,Y -333.698,Z 1501.517,A 0.000,B 0.000,C 90.000,E1 273.094} C_DIS
LIN {X 0.131,Y -320.305,Z 1501.515,A 0.000,B 0.000,C 90.000,E1 272.694} C_DIS
LIN {X 0.101,Y -308.765,Z 1501.514,A 0.000,B 0.000,C 90.000,E1 272.465} C_DIS
LIN {X 0.038,Y -296.361,Z 1501.513,A 0.000,B 0.000,C 90.000,E1 272.293} C_DIS
LIN {X -0.076,Y -287.382,Z 1501.512,A 0.000,B 0.000,C 90.000,E1 272.236} C_DIS
LIN {X -0.022,Y -277.243,Z 1501.512,A 0.000,B 0.000,C 90.000,E1 272.178} C_DIS
LIN {X -0.033,Y -181.235,Z 1501.512,A 0.000,B 0.000,C 90.000,E1 272.178} C_DIS
LIN {X 0.050,Y -181.575,Z 1501.501,A 0.000,B 0.000,C 90.000,E1 270.115} C_DIS
LIN {X 0.038,Y -180.877,Z 1501.473,A 0.000,B 0.000,C 90.000,E1 265.065} C_DIS
LIN {X -0.082,Y -178.996,Z 1501.444,A 0.000,B 0.000,C 90.000,E1 260.038} C_DIS
LIN {X 0.012,Y -178.582,Z 1501.440,A 0.000,B 0.000,C 90.000,E1 259.162} C_DIS
LIN {X -0.094,Y -175.635,Z 1501.411,A 0.000,B 0.000,C 90.000,E1 254.102} C_DIS
LIN {X -0.028,Y -172.354,Z 1501.388,A 0.000,B 0.000,C 90.000,E1 249.806} C_DIS
LIN {X -0.073,Y -171.138,Z 1501.378,A 0.000,B 0.000,C 90.000,E1 248.103} C_DIS
LIN {X -0.028,Y -167.443,Z 1501.354,A 0.000,B 0.000,C 90.000,E1 243.768} C_DIS
LIN {X 0.054,Y -166.839,Z 1501.349,A 0.000,B 0.000,C 90.000,E1 242.871} C_DIS
LIN {X -0.029,Y -162.822,Z 1501.325,A 0.000,B 0.000,C 90.000,E1 238.535} C_DIS
LIN {X 0.035,Y -161.508,Z 1501.315,A 0.000,B 0.000,C 90.000,E1 236.755} C_DIS
LIN {X -0.012,Y -157.506,Z 1501.291,A 0.000,B 0.000,C 90.000,E1 232.351} C_DIS
LIN {X 0.022,Y -155.527,Z 1501.276,A 0.000,B 0.000,C 90.000,E1 229.666} C_DIS
LIN {X 0.071,Y -151.825,Z 1501.251,A 0.000,B 0.000,C 90.000,E1 225.162} C_DIS
LIN {X 0.084,Y -150.040,Z 1501.236,A 0.000,B 0.000,C 90.000,E1 222.447} C_DIS
LIN {X -0.003,Y -146.856,Z 1501.211,A 0.000,B 0.000,C 90.000,E1 217.935} C_DIS
LIN {X 0.016,Y -145.440,Z 1501.196,A 0.000,B 0.000,C 90.000,E1 215.185} C_DIS
LIN {X 0.011,Y -142.861,Z 1501.170,A 0.000,B 0.000,C 90.000,E1 210.590} C_DIS
LIN {X 0.063,Y -141.477,Z 1501.149,A 0.000,B 0.000,C 90.000,E1 206.873} C_DIS
LIN {X -0.077,Y -139.380,Z 1501.113,A 0.000,B 0.000,C 90.000,E1 200.429} C_DIS
LIN {X 0.043,Y -138.833,Z 1501.098,A 0.000,B 0.000,C 90.000,E1 197.583} C_DIS
LIN {X -0.028,Y -138.353,Z 1501.056,A 0.000,B 0.000,C 90.000,E1 190.141} C_DIS
LIN {X -0.033,Y -139.525,Z 1501.004,A 0.000,B 0.000,C 90.000,E1 180.802} C_DIS
LIN {X 0.059,Y -141.195,Z 1500.973,A 0.000,B 0.000,C 90.000,E1 175.179} C_DIS
LIN {X 0.018,Y -142.571,Z 1500.958,A 0.000,B 0.000,C 90.000,E1 172.413} C_DIS
LIN {X -0.027,Y -144.859,Z 1500.932,A 0.000,B 0.000,C 90.000,E1 167.813} C_DIS
LIN {X -0.072,Y -147.485,Z 1500.912,A 0.000,B 0.000,C 90.000,E1 164.157} C_DIS
LIN {X -0.046,Y -150.072,Z 1500.892,A 0.000,B 0.000,C 90.000,E1 160.496} C_DIS
LIN {X -0.042,Y -153.421,Z 1500.871,A 0.000,B 0.000,C 90.000,E1 156.869} C_DIS
LIN {X 0.006,Y -156.842,Z 1500.851,A 0.000,B 0.000,C 90.000,E1 153.256} C_DIS
LIN {X 0.078,Y -160.922,Z 1500.832,A 0.000,B 0.000,C 90.000,E1 149.665} C_DIS
LIN {X 0.022,Y -163.046,Z 1500.822,A 0.000,B 0.000,C 90.000,E1 147.916} C_DIS
LIN {X 0.027,Y -167.440,Z 1500.802,A 0.000,B 0.000,C 90.000,E1 144.402} C_DIS
LIN {X -0.065,Y -171.277,Z 1500.788,A 0.000,B 0.000,C 90.000,E1 141.823} C_DIS
LIN {X -0.026,Y -176.170,Z 1500.769,A 0.000,B 0.000,C 90.000,E1 138.366} C_DIS
LIN {X -0.028,Y -180.442,Z 1500.754,A 0.000,B 0.000,C 90.000,E1 135.810} C_DIS
LIN {X -0.053,Y -185.847,Z 1500.736,A 0.000,B 0.000,C 90.000,E1 132.447} C_DIS
LIN {X 0.000,Y -190.470,Z 1500.722,A 0.000,B 0.000,C 90.000,E1 129.930} C_DIS
LIN {X -0.095,Y -196.222,Z 1500.703,A 0.000,B 0.000,C 90.000,E1 126.664} C_DIS
LIN {X 0.038,Y -201.354,Z 1500.689,A 0.000,B 0.000,C 90.000,E1 123.992} C_DIS
LIN {X 0.066,Y -201.830,Z 1500.687,A 0.000,B 0.000,C 90.000,E1 123.706} C_DIS
LIN {X 0.050,Y -315.735,Z 1500.687,A 0.000,B 0.000,C 90.000,E1 123.706} C_DIS
LIN {X -0.056,Y -316.949,Z 1500.687,A 0.000,B 0.000,C 90.000,E1 123.706} C_DIS
LIN {X -0.216,Y -320.879,Z 1500.686,A 0.000,B 0.000,C 90.000,E1 123.579} C_DIS
LIN {X 0.071,Y -323.099,Z 1500.685,A 0.000,B 0.000,C 90.000,E1 123.372} C_DIS
LIN {X 0.049,Y -326.978,Z 1500.683,A 0.000,B 0.000,C 90.000,E1 122.959} C_DIS
LIN {X 0.004,Y -328.868,Z 1500.682,A 0.000,B 0.000,C 90.000,E1 122.673} C_DIS
LIN {X -0.042,Y -330.352,Z 1500.680,A 0.000,B 0.000,C 90.000,E1 122.388} C_DIS
LIN {X 0.191,Y -345.256,Z 1500.659,A 0.000,B 0.000,C 90.000,E1 118.615} C_DIS
LIN {X -0.089,Y -357.969,Z 1500.644,A 0.000,B 0.000,C 90.000,E1 115.924} C_DIS
END
